// ---- DUTs/Sensirion/ST_SensirionFMStatus.TcDUT
TYPE ST_SensirionFMStatus :
STRUCT
	

	iFlowTicks	:	INT;
	uiSensorOutput	: UINT;
	iState	:	INT;
	rFlow	:	REAL; // units of uL/min
	xOoR	:	BOOL; // Out of range
	xFMMode :	BOOL; // calib mode 0 = prec, 1 = extended
	xFlowValid	:	BOOL; // driver completes successfully
	abReply	:	ARRAY[1..500] OF BYTE;
	bAdr	:	BYTE; //Device address
	bStatus	:	BYTE; //Sensor status
(* Bit 0: 0: Sensor idle
		1: Sensor Busy
Bit 1: 	0: Continuous Measurement disabled
		1: Continuous Measurement enabled
Bit 2: (for Firmware . 1.3)
		0: Auto detection Measurement disabled
		1: Auto detection Measurement enabled
Bit 3: (for Firmware . 1.3)
		0: No Auto Measurement since last read out Status
		1: Auto Measurement finished since last read out Status, is set back to 0 after read out *)

END_STRUCT
END_TYPE

// ---- DUTs/ST_M3GasManifold.TcDUT
TYPE ST_M3GasManifold :
STRUCT
	stManiVlv1	:	ST_ManifoldValve;
	stManiVlv2	:	ST_ManifoldValve;
	stManiVlv3	:	ST_ManifoldValve;
	stManiVlv4	:	ST_ManifoldValve;
	stManiVlv5	:	ST_ManifoldValve;
	stManiVlv6	:	ST_ManifoldValve;
	stManiVlv7	:	ST_ManifoldValve;
	stManiVlv8	:	ST_ManifoldValve;
	
	xOnline	:	BOOL; //WC inverse (true is good)
END_STRUCT
END_TYPE

// ---- DUTs/ST_Proportionair.TcDUT
TYPE ST_Proportionair :
STRUCT
	
(* Control *)
xEnable	:	BOOL;
iSetpoint	:	INT;
iSetpointRaw	:	INT;
iHiLimit	:	INT;
iLoLimit	:	INT;

(* Readback *)
xStable	:	BOOL;//TTL signal from the proportionair controller that the pressure is stable
iPressure	:	INT;
iPressureRaw : INT;


END_STRUCT
END_TYPE

// ---- DUTs/ST_Selector.TcDUT
TYPE ST_Selector :
STRUCT

	(* Meta info *)
	iId	: INT;	// Used to ID the selector attached to the system
	(* iId: Implemented to support switching selectors on the fly,
	the ID tells us which flow meter code to use, as the M2
	used several different flowmeters. *)

	(* Flowmeter *)
	(* Declare a structure for every possible FM *)
	stSelFMStatusBh	:	ST_BhFMStatus;
	stSelFMStatusSens	:	ST_SensirionFMStatus;
	stSelFMControlBh	:	ST_BhFMControl;
	stSelFMControlSens	:	ST_SensirionFMControl;
		
	
	//Common parameters
	iFlowMeterType	:	INT; //see below
	(*  1 = Sensirion
		2 = Bronkhorst
	*)
	
	xFMReset : BOOL; // Pulse only.
	rFlow : REAL; //uL/min
	xFMOoR	:	BOOL; // Out of range (too high)
	xFlowValid	:	BOOL; // driver completes successfully
	xFMModeReq	:	BOOL; //for sensirion calibration range (request)
	xFMModeRb	:	BOOL; //for sensirion calibration range (readback)
	(*
	field(ZRST, "OK")
	field(ONST, "OoR>")
	field(TWST, "<OoR")
	field(THST, "Flow Invalid")
	*)
	iFMState	:	INT;

	(* Selector controls *)
	xResLock	:	BOOL; // request to lock the valves
	xResUnlock	:	BOOL; // request to unlock the valves
	xResLocked	:	BOOL; // valve movement is locked
	xResSyncd	:	BOOL; // valves are on the same position
	iSyncReqPos	:	INT;
	iVici1ReqPos : INT;
	iVici2ReqPos : INT;
	stViciVlvCtrl	: ARRAY[1..2] OF	ST_ViciControl;
	
	
	(* Selector Readbacks *)
	iSyncResPos : INT;
	stViciVlvStatus	: ARRAY[1..2] OF	ST_ViciStatus;
	
	(* Shakers *)
	stShaker01	:	ST_Shaker;
	stShaker02	:	ST_Shaker;
	stShaker03	:	ST_Shaker;
	stShaker04	:	ST_Shaker;
	

END_STRUCT
END_TYPE

// ---- DUTs/ST_ShakerControls.TcDUT
TYPE ST_ShakerControls :
STRUCT
	
xShaker1On	:	BOOL;
xShaker2On	:	BOOL;
xShaker3On	:	BOOL;
xShaker4On	:	BOOL;
xShaker5On	:	BOOL;
xShaker6On	:	BOOL;
xShaker7On	:	BOOL;
xShaker8On	:	BOOL;

END_STRUCT
END_TYPE

// ---- DUTs/Vici/ST_ViciControl.TcDUT
TYPE ST_ViciControl :
STRUCT
	sViciReply			: STRING;
	iReqPos				: INT;
	xDirection			:BOOL;
	iAddress				:INT;
END_STRUCT
END_TYPE

// ---- GVLs/GVL.TcGVL
VAR_GLOBAL
 mb_Input_Coils   : ARRAY [0..255] OF BOOL;
 mb_Output_Coils : ARRAY [0..255] OF BOOL;
 mb_Input_Registers : ARRAY [0..255] OF WORD;
 mb_Output_Registers : ARRAY [0..255] OF WORD;
 
 mb_PLC_Memory	AT	%MW0	:	ARRAY[0..1000] OF WORD;
 
 	g_xFirstPass: BOOL := TRUE;
	g_xIOState	:	BOOL := FALSE;
	g_aEcatMaster1 AT %I* : AMSNETID;
	g_aEcatMaster2 AT %I* : AMSNETID;
	

 
END_VAR

// ---- GVLs/GVL_Autosave.TcGVL
VAR_GLOBAL PERSISTENT
	
	gp_stWaterRegDeadband	:	ST_RegDeadbandControls;
	gp_stSheathRegDeadband	:	ST_RegDeadbandControls;

	gp_stSelector	:	ST_Selector;
	gp_stSelector2	:	ST_Selector;
	
	gp_stRegProp1	:	ST_Proportionair;
	gp_stRegProp2	:	ST_Proportionair;
	gp_stRegProp3	:	ST_Proportionair;
	gp_stRegProp4	:	ST_Proportionair;

END_VAR

// ---- GVLs/GVL_ComBuffers.TcGVL
VAR_GLOBAL
	
	SerialRXBuffer_SelVici : ComBuffer;
	SerialTXBuffer_SelVici : ComBuffer;
	
	SerialRXBuffer_SelFlwMtr : ComBuffer;
	SerialTXBuffer_SelFlwMtr : ComBuffer;
	
	SerialRXBuffer_Sel2FlwMtr : ComBuffer;
	SerialTXBuffer_Sel2FlwMtr : ComBuffer;
	
	SerialRXBuffer_Sel2Vici : ComBuffer;
	SerialTXBuffer_Sel2Vici : ComBuffer;
	
	SerialRXBuffer_CoolerShakerTEC : ComBuffer;
	SerialTXBuffer_CoolerShakerTEC : ComBuffer;
	
END_VAR

// ---- GVLs/GVL_Devices.TcGVL
VAR_GLOBAL
	
	(* Selector*)
	stSelector	:	ST_Selector;
	stSelector2	:	ST_Selector;
	
	(* Cooler shaker *)
	stTECCtrl	: ARRAY[1..3] OF	ST_TECControl;
	stTECStatus	: ARRAY[1..3] OF	ST_TECStatus;
	
	stRegProp1	:	ST_Proportionair;
	stRegProp2	:	ST_Proportionair;
	stRegProp3	:	ST_Proportionair;
	stRegProp4	:	ST_Proportionair;
	
	(* Shakers *)
	stShaker01	:	ST_Shaker;
	stShaker02	:	ST_Shaker;
	stShaker03	:	ST_Shaker;
	stShaker04	:	ST_Shaker;
	
	(* Minitti Manifold *)
	stGasMani	:	ST_M3GasManifold;
	
	(* ALI *)
	stALI	:	ST_ALI;

END_VAR

// ---- GVLs/GVL_IO.TcGVL
VAR_GLOBAL
	
	iq_stM2SelectorA	:	ST_M2SelectorIO;
	iq_stM2SelectorB	:	ST_M2SelectorIO;

	iq_stM3SelectorA	:	ST_M3SelectorIO;
	iq_stM3SelectorB	:	ST_M3SelectorIO;
	
	iq_stPressCtrlA		:	ST_M3PressCtrlIO;
	iq_stPressCtrlB		:	ST_M3PressCtrlIO;

	i_iFscEB1Ch0AI	AT	%I*	:	INT;
	i_iFscEB1Ch1AI	AT	%I*	:	INT;
	i_iFscEB1Ch2AI	AT	%I*	:	INT;
	i_iFscEB1Ch3AI	AT	%I*	:	INT;
	
	iq_stM3GasManifold	:	ST_M3GasManifoldIO;

END_VAR

// ---- Version/Global_Version.TcGVL
// This function has been automatically generated from the project information.
VAR_GLOBAL CONSTANT
	{attribute 'const_non_replaced'}
	stLibVersion_SDS_M2 : ST_LibVersion := (iMajor := 2, iMinor := 6, iBuild := 0, iRevision := -1, sVersion := '2.6.0');
END_VAR

// ---- POUs/MAIN.TcPOU
PROGRAM MAIN
VAR
	
		fb_S_UPS	:	FB_S_UPS;
		
		fbEcatDiag1	:	FB_EcatDiag;
		fbEcatDiag2 :	FB_EcatDiag;
	
END_VAR



//fb_S_UPS.iPLCPort := AMSPORT_R0_PLC_RTS2;
fb_S_UPS(iPLCPort:=851);


p_modbusRx();

p_Autosave();

p_ESTOP();

fbEcatDiag1(i_AMSNetId:=g_aEcatMaster1, i_xFirstPass:=g_xFirstPass, q_xAllStatesGood=>g_xIOState);
fbEcatDiag2(i_AMSNetId:=g_aEcatMaster2, i_xFirstPass:=g_xFirstPass, q_xAllStatesGood=>g_xIOState);

p_SoftIO();

//p_SelectorDetector();

p_SampleSelector();
p_SampleSelector2();
p_Regulators();
p_Manifold();
p_ALI();
//p_VacGaugeSup();


//p_CoolerShaker();

p_ModbusTx();

p_StatusLights();

(* Following execution of all the programs, set the first pass false *)
g_xFirstPass := FALSE;

END_PROGRAM

// ---- POUs/p_ModbusRx.TcPOU
PROGRAM p_ModbusRx
VAR
END_VAR

(* Modbus Controls from EPICS *)

(* General System Controls *)
xEnableRemoteControl := mb_Output_Coils[0];
g_xEstop		:= mb_Output_Coils[1];

IF xEnableRemoteControl THEN
xN2Purge	:= mb_Output_Coils[9];

(* Selector Controls *)
stSelector.iVici1ReqPos := mb_Output_Registers[30];
stSelector.iVici2ReqPos := mb_Output_Registers[31];
stSelector.iSyncReqPos	:= mb_Output_Registers[32];

stSelector.xResLock := mb_Output_Coils[30];
stSelector.xFMReset := mb_Output_Coils[31];
stSelector.xFMModeReq 	:= mb_Output_Coils[32];
stSelector.xResUnlock := mb_Output_Coils[33];

stSelector.stShaker01.i_xEpics := mb_Output_Coils[10];
stSelector.stShaker02.i_xEpics := mb_Output_Coils[11];
stSelector.stShaker03.i_xEpics := mb_Output_Coils[12];
stSelector.stShaker04.i_xEpics := mb_Output_Coils[13];

(* Selector 2 Controls *)
stSelector2.iVici1ReqPos := mb_Output_Registers[40];
stSelector2.iVici2ReqPos := mb_Output_Registers[41];
stSelector2.iSyncReqPos	:= mb_Output_Registers[42];

stSelector2.xResLock := mb_Output_Coils[40];
stSelector2.xFMReset := mb_Output_Coils[41];
stSelector2.xFMModeReq 	:= mb_Output_Coils[42];
stSelector2.xResUnlock := mb_Output_Coils[43];

stSelector2.stShaker01.i_xEpics := mb_Output_Coils[44];
stSelector2.stShaker02.i_xEpics := mb_Output_Coils[45];
stSelector2.stShaker03.i_xEpics := mb_Output_Coils[46];
stSelector2.stShaker04.i_xEpics := mb_Output_Coils[47];

(* Proportionair controls *)
stRegProp1.xEnable:=mb_Output_Coils[50];  //Proportionair controls
stRegProp2.xEnable:=mb_Output_Coils[51];  //Proportionair controls

stRegProp3.xEnable:=mb_Output_Coils[52];  //Proportionair controls
stRegProp4.xEnable:=mb_Output_Coils[53];  //Proportionair controls

stRegProp1.iSetpoint:=mb_Output_Registers[50];  //Proportionair controls
stRegProp2.iSetpoint:=mb_Output_Registers[51];  //Proportionair controls
stRegProp1.iHiLimit:=mb_Output_Registers[52];  //Proportionair controls
stRegProp2.iHiLimit:=mb_Output_Registers[53];  //Proportionair controls

stRegProp3.iSetpoint:=mb_Output_Registers[54];  //Proportionair controls
stRegProp4.iSetpoint:=mb_Output_Registers[55];  //Proportionair controls
stRegProp3.iHiLimit:=mb_Output_Registers[56];  //Proportionair controls
stRegProp4.iHiLimit:=mb_Output_Registers[57];  //Proportionair controls

(* Digital output controls *)
stManiVlv1.xSW:=mb_Output_Coils[60];  //Minitti manifold valve controls
stManiVlv2.xSW:=mb_Output_Coils[61];  //Minitti manifold valve controls
stManiVlv3.xSW:=mb_Output_Coils[62];  //Minitti manifold valve controls
stManiVlv4.xSW:=mb_Output_Coils[63];  //Minitti manifold valve controls
stManiVlv5.xSW:=mb_Output_Coils[64];  //Minitti manifold valve controls
stManiVlv6.xSW:=mb_Output_Coils[65];  //Minitti manifold valve controls
stManiVlv7.xSW:=mb_Output_Coils[66];  //Minitti manifold valve controls
stManiVlv8.xSW:=mb_Output_Coils[67];  //Minitti manifold valve controls
//=========================================================
// ALI Controls
	stALI.axisX.xStart:=mb_Output_Coils[80];  //ALI_Manip
	stALI.axisX.xStop:=mb_Output_Coils[81];  //ALI_Manip
	stALI.axisY.xStart:=mb_Output_Coils[82];  //ALI_Manip
	stALI.axisY.xStop:=mb_Output_Coils[83];  //ALI_Manip
	stALI.axisZ.xStart:=mb_Output_Coils[84];  //ALI_Manip
	stALI.axisZ.xStop:=mb_Output_Coils[85];  //ALI_Manip
	
	stALI.stPropVlv.xEnable := mb_Output_Coils[86];
	
	stALI.axisX.xReset:=mb_Output_Coils[87];  //ALI_Manip
	stALI.axisY.xReset:=mb_Output_Coils[88];  //ALI_Manip
	stALI.axisZ.xReset:=mb_Output_Coils[89];  //ALI_Manip
	
	stALI.stPropVlv.i_iPercOpenSP := mb_Output_Registers[80]; //ALI Propvalve
	stALI.stPropVlv.ePVCtrlStateReq := mb_Output_Registers[81]; //ALI Propvalve
	MEMCPY(srcAddr:=ADR(mb_PLC_Memory[90]), destAddr:=ADR(stALI.axisX.rReqAbsPos), n:=SIZEOF(stALI.axisX.rReqAbsPos)); //ALI CTRL
	MEMCPY(srcAddr:=ADR(mb_PLC_Memory[92]), destAddr:=ADR(stALI.axisY.rReqAbsPos), n:=SIZEOF(stALI.axisY.rReqAbsPos)); //ALI CTRL
	MEMCPY(srcAddr:=ADR(mb_PLC_Memory[94]), destAddr:=ADR(stALI.axisZ.rReqAbsPos), n:=SIZEOF(stALI.axisZ.rReqAbsPos)); //ALI CTRL
	MEMCPY(srcAddr:=ADR(mb_PLC_Memory[96]), destAddr:=ADR(stALI.stPropVlv.i_rPressSP), n:=SIZEOF(stALI.stPropVlv.i_rPressSP)); //ALI CTRL

END_IF

END_PROGRAM

// ---- POUs/p_Autosave.TcPOU
PROGRAM p_Autosave
VAR
END_VAR

(* If first pass, copy all persistent variables (which should be intialized to old values) back into the operational variables *)
IF g_xFirstPass THEN
	
	stRegProp1 := gp_stRegProp1;
	stRegProp2 := gp_stRegProp2;
	stRegProp3 := gp_stRegProp3;
	stRegProp4 := gp_stRegProp4;
	
ELSE
	gp_stRegProp1 := stRegProp1;
	gp_stRegProp2 := stRegProp2;
	gp_stRegProp3 := stRegProp3;
	gp_stRegProp4 := stRegProp4;
	
END_IF

END_PROGRAM

// ---- POUs/p_ESTOP.TcPOU
PROGRAM p_ESTOP
VAR
	rtEstop : R_TRIG;
END_VAR

(* 
Estop checks for a rising edge on the estop global variable then triggeres the following actions
1. Set selector to position 12, the default resting place
2. Set the water regulator to 0
The sheath regulator is not set to zero at this point because we don't want to ice the jet.
*)

rtEstop(CLK:=g_xEstop);

(* Check for E-Stop *)
IF rtEstop.Q THEN
	stSelector.iVici1ReqPos := 12;
	stSelector.iVici2ReqPos := 12;
	stSelector.iSyncReqPos	:= 12;	
END_IF

END_PROGRAM

// ---- POUs/p_SoftIO.TcPOU
PROGRAM p_SoftIO
VAR
END_VAR

(* Shakers *)
stSelector.stShaker01.i_xSwitch := iq_stM2SelectorA.i_EP2338_Ch5;
stSelector.stShaker02.i_xSwitch := iq_stM2SelectorA.i_EP2338_Ch6;
stSelector.stShaker03.i_xSwitch := iq_stM2SelectorA.i_EP2338_Ch7;
stSelector.stShaker04.i_xSwitch := iq_stM2SelectorA.i_EP2338_Ch8;

iq_stM2SelectorA.q_EP2338_Ch1	:= stSelector.stShaker01.q_xPwrDO;
iq_stM2SelectorA.q_EP2338_Ch2	:= stSelector.stShaker02.q_xPwrDO;
iq_stM2SelectorA.q_EP2338_Ch3	:= stSelector.stShaker03.q_xPwrDO;
iq_stM2SelectorA.q_EP2338_Ch4	:= stSelector.stShaker04.q_xPwrDO;

stSelector2.stShaker01.i_xSwitch := iq_stM2SelectorB.i_EP2338_Ch5;
stSelector2.stShaker02.i_xSwitch := iq_stM2SelectorB.i_EP2338_Ch6;
stSelector2.stShaker03.i_xSwitch := iq_stM2SelectorB.i_EP2338_Ch7;
stSelector2.stShaker04.i_xSwitch := iq_stM2SelectorB.i_EP2338_Ch8;

iq_stM2SelectorB.q_EP2338_Ch1	:= stSelector2.stShaker01.q_xPwrDO;
iq_stM2SelectorB.q_EP2338_Ch2	:= stSelector2.stShaker02.q_xPwrDO;
iq_stM2SelectorB.q_EP2338_Ch3	:= stSelector2.stShaker03.q_xPwrDO;
iq_stM2SelectorB.q_EP2338_Ch4	:= stSelector2.stShaker04.q_xPwrDO;

stRegProp1.iPressureRaw := iq_stPressCtrlA.i_EP4374_Ch1;
stRegProp2.iPressureRaw := iq_stPressCtrlA.i_EP4374_Ch2;

iq_stPressCtrlA.q_EP4374_Ch3 := stRegProp1.iSetpointRaw;
iq_stPressCtrlA.q_EP4374_Ch4 := stRegProp2.iSetpointRaw;

stRegProp3.iPressureRaw := iq_stPressCtrlB.i_EP4374_Ch1;
stRegProp4.iPressureRaw := iq_stPressCtrlB.i_EP4374_Ch2;

iq_stPressCtrlB.q_EP4374_Ch3 := stRegProp3.iSetpointRaw;
iq_stPressCtrlB.q_EP4374_Ch4 := stRegProp4.iSetpointRaw;

END_PROGRAM

// ---- POUs/p_Regulators.TcPOU
PROGRAM p_Regulators
VAR

fbRegProp1	:	FB_ProportionairRegulator;
fbRegProp2	:	FB_ProportionairRegulator;
fbRegProp3	:	FB_ProportionairRegulator;
fbRegProp4	:	FB_ProportionairRegulator;

END_VAR

(* Proportionair regulators *)
fbRegProp1(iq_stRegProp:=stRegProp1);
fbRegProp2(iq_stRegProp:=stRegProp2);
fbRegProp3(iq_stRegProp:=stRegProp3);
fbRegProp4(iq_stRegProp:=stRegProp4);

END_PROGRAM

// ---- POUs/Regulators/FB_ProportionairRegulator.TcPOU
FUNCTION_BLOCK FB_ProportionairRegulator
VAR_INPUT
END_VAR
VAR_OUTPUT
END_VAR
VAR_IN_OUT
	iq_stRegProp	:	ST_Proportionair;
END_VAR
VAR
END_VAR

(* A. Wallace 2015-10-7
Proportionair regulator control *)

(* Pressure signal conversion, max pressure out 1000 (I think...) *)
iq_stRegProp.iPressure := REAL_TO_INT(1000 * (INT_TO_REAL(iq_stRegProp.iPressureRaw) / 32767));

iq_stRegProp.iSetpoint := LIMIT(iq_stRegProp.iLoLimit, iq_stRegProp.iSetpoint, iq_stRegProp.iHiLimit);

iq_stRegProp.iSetpointRaw := REAL_TO_INT( (INT_TO_REAL(iq_stRegProp.iSetpoint)/1000)*32767);

END_FUNCTION_BLOCK

// ---- POUs/p_Manifold.TcPOU
PROGRAM p_Manifold
VAR
	fbManiValve : FB_ManiValve;
END_VAR

(* Valve 1 *)
stManiVlv1.xILK := TRUE;
fbManiValve(iq_valve:=stManiVlv1);

(* Valve 2 *)
stManiVlv2.xILK := TRUE;
fbManiValve(iq_valve:=stManiVlv2);

(* Valve 3 *)
stManiVlv3.xILK := TRUE;
fbManiValve(iq_valve:=stManiVlv3);

(* Valve 4 *)
stManiVlv4.xILK := TRUE;
fbManiValve(iq_valve:=stManiVlv4);

(* Valve 5 *)
stManiVlv5.xILK := TRUE;
fbManiValve(iq_valve:=stManiVlv5);

(* Valve 6 *)
stManiVlv6.xILK := TRUE;
fbManiValve(iq_valve:=stManiVlv6);

(* Valve 7 *)
stManiVlv7.xILK := TRUE;
fbManiValve(iq_valve:=stManiVlv7);

(* Valve 8 *)
stManiVlv8.xILK := TRUE;
fbManiValve(iq_valve:=stManiVlv8);

END_PROGRAM

// ---- POUs/p_ALI.TcPOU
PROGRAM p_ALI
VAR
	fbALI_A	:	FB_ALI;
END_VAR

fbALI_A(iq_Injector:=stALI);

END_PROGRAM

// ---- POUs/ALI/FB_ALI.TcPOU
FUNCTION_BLOCK FB_ALI
VAR_IN_OUT
	iq_Injector	:	ST_ALI;
END_VAR
VAR_INPUT
END_VAR
VAR_OUTPUT
END_VAR
VAR
	fb925ALINB1 : FB_925;
	fb925ALINB2 : FB_925;
	fb722ALINB3 : FB_GCM;
	
	fbManipX	:	FB_ManipAxis;
	fbManipY	:	FB_ManipAxis;
	fbManipZ	:	FB_ManipAxis;
	

	
	fbPropValve		:	FB_PropValve;
	
	ftHotPlug	:	F_TRIG;
END_VAR

//When the system is plugged in, WC goes to zero, so reset motion control and other stuff
ftHotPlug(CLK:=iq_Injector.i_SyncUnitWC);

(* Soft IO *)
iq_Injector.stNozzleBoxVG.iPRESS_R :=iq_Injector.i_EP3174_Ch1;
iq_Injector.stSkimmerVG.iPRESS_R := iq_Injector.i_EP3174_Ch2;
iq_Injector.stRelaxVG.iPRESS_R := iq_Injector.i_EP3174_Ch3;

(* Vacuum Gauge Supervisor *)
fb925ALINB1(VG:=iq_Injector.stNozzleBoxVG);
fb925ALINB2(VG:=iq_Injector.stSkimmerVG);
fb722ALINB3(VG:=iq_Injector.stRelaxVG);

(* Butterfly valve *)
iq_Injector.stPropVlv.xInterlock := TRUE;
fbPropValve(stPropValve:=iq_Injector.stPropVlv, i_xExtIlk := TRUE);

(* Manipulator *)
fbManipX(iq_ManipAxis:=iq_Injector.axisX, i_xHotPlug:=ftHotPlug.Q);
fbManipY(iq_ManipAxis:=iq_Injector.axisY, i_xHotPlug:=ftHotPlug.Q);
fbManipZ(iq_ManipAxis:=iq_Injector.axisZ, i_xHotPlug:=ftHotPlug.Q);
F_AxisRef_To_MSTA(stManipAxis:=iq_Injector.axisX, MSTA=>iq_Injector.axisX.uiMsta);
F_AxisRef_To_MSTA(stManipAxis:=iq_Injector.axisY, MSTA=>iq_Injector.axisY.uiMsta);
F_AxisRef_To_MSTA(stManipAxis:=iq_Injector.axisZ, MSTA=>iq_Injector.axisZ.uiMsta);

END_FUNCTION_BLOCK

// ---- POUs/ALI/FB_ManipAxis.TcPOU
FUNCTION_BLOCK FB_ManipAxis
VAR_INPUT
	i_xHotPlug	:	BOOL;
END_VAR
VAR_OUTPUT
	q_asResult: ARRAY [1..20] OF STRING;
	q_xError	:	BOOL;
END_VAR
VAR_IN_OUT
	iq_ManipAxis	:	ST_ManipAxis;
END_VAR
VAR

	mcPower	:	MC_Power;
	mcReset	:	MC_Reset;
	mcMoveAbsolute : ARRAY[1..2] OF MC_MoveAbsolute;
	mcHalt	:	MC_Halt;
	mcSmoothMover	:	MC_SmoothMover;
	//Error Stuff
	indexResult: INT := 1;
	fbFormatString	:	FB_FormatString;
	
	xInitComplete	:	BOOL := FALSE;
	
	imcBlockIndex: INT;
	
	rtEnable : R_TRIG;
	ftEnable : F_TRIG;
	rtStop	:	R_TRIG;
	rtStart	:	R_TRIG;
	rReqAbsPosOld: REAL := 0;
	rReqAbsPosPrevious: REAL;
	iI: INT;
END_VAR

(* Manipulator Axis Function Block
Alex Wallace, 2016-8-8 

This block works by jumping between two absolute move blocks and buffering
the motion between them.
*)


rtEnable(CLK:=iq_ManipAxis.xEnable);
ftEnable(CLK:=iq_ManipAxis.xEnable);

//Update status
iq_ManipAxis.stAxis();

IF rtEnable.Q OR ftEnable.Q THEN
	xInitComplete := FALSE;
	iq_ManipAxis.eState := Init;
ELSIF xInitComplete THEN
	iq_ManipAxis.eState := MoveEnabled;
END_IF

//For EPICS, because the modbus map was made for 32 bit..
iq_ManipAxis.rActPos := LREAL_TO_REAL(iq_ManipAxis.stAxis.NcToPlc.ActPos);


CASE iq_ManipAxis.eState OF
	0: iq_ManipAxis.eState := Init;
	Init:
	(* Start by initializing the motor axis *)
	mcPower.Enable := iq_ManipAxis.xEnable;
	iq_ManipAxis.rReqAbsPos := iq_ManipAxis.rActPos; //do this when the PLC comes up so we don't just lose the position if we tweak
	IF mcPower.Status THEN //success
		xInitComplete := TRUE;
		q_asResult[indexResult] := 'Motor init success';
		indexResult := indexResult + 1;
		iq_ManipAxis.eState := MoveEnabled;
	ELSIF mcPower.Error THEN
		mcPower.Enable := FALSE;
		fbFormatString(sFormat:='Init mcPower Error: %s', arg1:=F_UDINT(mcPower.ErrorID));
		ActError();
	END_IF
		
	MoveEnabled:
		mcSmoothMover.Enable := iq_ManipAxis.xEnable;
		mcSmoothMover.ReqAbsPos := LIMIT(-100, REAL_TO_LREAL(iq_ManipAxis.rReqAbsPos), 100);
		mcSmoothMover.Execute := iq_ManipAxis.xStart;
		(*We've already captured the rising edge of start (if there was one, so 
		go ahead and reset it.*)
		iq_ManipAxis.xStart := FALSE;
		
		//Halt
		mcHalt.Execute S= iq_ManipAxis.xStop;
		mcHalt.Execute R= mcHalt.Busy;
		iq_ManipAxis.xStop R= mcHalt.Busy;
		IF mcPower.Error OR mcSmoothMover.Error THEN
			iq_ManipAxis.eState:=Error;
		END_IF
		
	Error:
		mcReset.Execute := rtEnable.Q OR i_xHotPlug OR iq_ManipAxis.xReset;
		IF mcReset.Done THEN
			q_xError := FALSE;
			mcReset.Execute := FALSE;
			iq_ManipAxis.xReset := FALSE;
			iq_ManipAxis.eState:=Init;
		END_IF
	
END_CASE


(* Run the mc blocks *)
ActPower();
mcReset(Axis:=iq_ManipAxis.stAxis);
mcSmoothMover(Axis:=iq_ManipAxis.stAxis,
	Velocity:=iq_ManipAxis.lrVelocity);
mcHalt(Axis:=iq_ManipAxis.stAxis);

iq_ManipAxis.xDmov := mcHalt.Done OR mcSmoothMover.Done;
iq_ManipAxis.xMovn := mcHalt.Busy OR mcSmoothMover.Busy;

//For display, this logic is not for safety
iq_ManipAxis.xHLS := NOT iq_ManipAxis.xHiLS;
iq_ManipAxis.xLLS := NOT iq_ManipAxis.xLoLS;

ACTION ActPower:
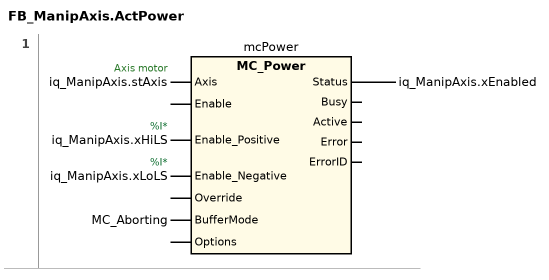
// NETWORK 1
//   iq_ManipAxis.stAxis: Axis motor
//   iq_ManipAxis.xHiLS: AT %I*
//   iq_ManipAxis.xLoLS: AT %I*
mcPower(
    Axis := iq_ManipAxis.stAxis,
    Enable_Positive := iq_ManipAxis.xHiLS,
    Enable_Negative := iq_ManipAxis.xLoLS,
    BufferMode := MC_Aborting); // MC_Power
iq_ManipAxis.xEnabled := mcPower.Status;
END_ACTION

ACTION ActError:
(* Error action
*)

//Reset the debugging index
IF indexResult > 20 THEN indexResult := 1; END_IF

iq_ManipAxis.eState := Error;
q_xError	:=	TRUE;
q_asResult[indexResult] := fbFormatString.sOut;
indexResult := indexResult +1;
END_ACTION

END_FUNCTION_BLOCK

// ---- POUs/ALI/MC_SmoothMover.TcPOU
FUNCTION_BLOCK MC_SmoothMover
VAR_IN_OUT
	Axis	:	AXIS_REF;
END_VAR
VAR_INPUT
	Velocity : LREAL;
	ReqAbsPos : LREAL; //A
	Enable	:	BOOL; //While true the block will accept new positions and attempt to move to them if they are different
	Execute	:	BOOL; //Will retry a move if the target position is the same
END_VAR
VAR_OUTPUT
	Done	:	BOOL;
	Busy	:	BOOL;
	Error	:	BOOL;
END_VAR
VAR
	mcMoveAbsolute : ARRAY[1..2] OF MC_MoveAbsolute;
	iI: INT;
	imcBlockIndex: INT;
	ReqAbsPosPrevious	: LREAL;
	rtExecute: R_TRIG;
END_VAR

(* Smooth Mover
2017-8-30
A. Wallace

Enable means the block will always aquire new positions as they are updated. Execute
can be used to retry a move.
*)


rtExecute(CLK:=Execute);

IF ( (ReqAbsPos <> ReqAbsPosPrevious AND Enable) OR rtExecute.Q) THEN
			mcMoveAbsolute[imcBlockIndex].Execute := FALSE;
			imcBlockIndex := imcBlockIndex + 1;
			IF imcBlockIndex >2 THEN imcBlockIndex := 1; END_IF
			mcMoveAbsolute[imcBlockIndex].Position := ReqAbsPos;
			mcMoveAbsolute[imcBlockIndex].Execute := TRUE;
			ReqAbsPosPrevious := ReqAbsPos;
		ELSIF mcMoveAbsolute[imcBlockIndex].Done OR 
				mcMoveAbsolute[imcBlockIndex].CommandAborted OR 
				mcMoveAbsolute[imcBlockIndex].Busy OR 
				mcMoveAbsolute[imcBlockIndex].Error THEN
			mcMoveAbsolute[imcBlockIndex].Execute := FALSE;
		END_IF
		
FOR iI := 1 TO 2 DO
	mcMoveAbsolute[iI](Axis := Axis, Velocity:=Velocity, BufferMode:=MC_Aborting);
END_FOR

Error := mcMoveAbsolute[1].Error OR mcMoveAbsolute[2].Error;
Done S= mcMoveAbsolute[1].Done OR mcMoveAbsolute[2].Done;
Busy := mcMoveAbsolute[1].Busy OR mcMoveAbsolute[2].Busy;
Done R= Busy OR Error;

END_FUNCTION_BLOCK

// ---- POUs/ALI/FB_PropValve.TcPOU
FUNCTION_BLOCK FB_PropValve
VAR_INPUT
	i_xExtIlk	:	BOOL;
END_VAR
VAR_OUTPUT
	q_xError	:	BOOL;
END_VAR
VAR_IN_OUT
	stPropValve	:	ST_PropValveMKS253;
END_VAR
VAR
	xInterlock	:	BOOL;
	
	eState : E_PropValveFBState := E_PropValveFBState.Init;
	stDiag	:	ST_fbDiagnostics;
	
	mcPower	:	MC_Power;
	mcJog	:	MC_Jog;
	mcReset	:	MC_Reset;
	mcSmoothMover	:	MC_SmoothMover;
	tofLLSFilter	:	TOF := (PT:=T#100MS);
	tofHLSFilter	:	TOF := (PT:=T#100MS);
	
	fbPID	:	FB_PID_EXT;
	
	AnyError: BOOL;
	xReady	:	BOOL;
	rtReset: R_TRIG;
	
	UpperLimit : LREAL := 2000;
END_VAR

(* Provide the motor enable and limit switch functions for the MKS 253 valve *)

xInterlock := stPropValve.xInterlock AND i_xExtIlk;
stPropValve.xEnable R= NOT xInterlock;


rtReset(CLK:=stPropValve.xEnable);

(* The low limit switch was flakey, I added the filters *)
tofLLSFilter(IN:=stPropValve.i_LLS);
tofHLSFilter(IN:=stPropValve.i_HLS);
mcPower.Enable_Positive := tofHLSFilter.Q;
mcPower.Enable_Negative := tofLLSFilter.Q;
mcPower.Enable := xInterlock AND stPropValve.xEnable;
stPropValve.xEnabled := mcPower.Enable;
(* Move the valve *)

IF AnyError THEN
	eState := E_PropValveFBState.Error;
	stPropValve.ePVCtrlStateReq := HMI_PropValveCtrlState.Hold;
ELSIF xReady THEN
	CASE stPropValve.ePVCtrlStateReq OF
		HMI_PropValveCtrlState.Hold:
			eState := E_PropValveFBState.Hold;
		HMI_PropValveCtrlState.Manual:
			eState := E_PropValveFBState.Manual;
		HMI_PropValveCtrlState.Pressure:
			eState := E_PropValveFBState.Pressure;
	END_CASE
ELSE
	eState := E_PropValveFBState.Init;
END_IF

CASE eState OF
	E_PropValveFBState.Init:
		//This state is reached at startup and after a reset
		//It seeks the closed limit switch and moves to hold
		stPropValve.ePVCtrlState := HMI_PropValveCtrlState.Hold;
		fbPID.i_Reset := TRUE;
		IF NOT tofLLSFilter.Q AND mcPower.Status THEN
			stPropValve.ePVCtrlStateReq := HMI_PropValveCtrlState.Hold;
			fbPID.i_Reset := TRUE;
			xReady := TRUE;
		END_IF
	E_PropValveFBState.Hold:
		stPropValve.ePVCtrlState := HMI_PropValveCtrlState.Hold;
		mcJog.JogForward := FALSE;
		mcJog.JogBackwards := FALSE;
		fbPID.i_Hold := TRUE;
		
	E_PropValveFBState.Pressure:
		stPropValve.ePVCtrlState := HMI_PropValveCtrlState.Pressure;
		
		fbPID.i_Hold := FALSE;
		fbPID.i_Reset := FALSE;
		
		//If the PID output is positive, jog forward, velocity scaled by the PID output
		//likewise for a negative PID output
		mcJog.JogForward := fbPID.q_lrCtrlOutput > 0;
		mcJog.JogBackwards := fbPID.q_lrCtrlOutput < 0;
		mcJog.Velocity := ABS(fbPID.q_lrCtrlOutput) * stPropValve.lrMaxSpeed;
		
	E_PropValveFBState.Manual:
		stPropValve.ePVCtrlState := HMI_PropValveCtrlState.Manual;
		fbPID.i_Hold := TRUE;
		mcSmoothMover.Enable := TRUE;
		mcSmoothMover.ReqAbsPos := LIMIT(0, INT_TO_LREAL(stPropValve.i_iPercOpenSP), 100)/100*UpperLimit;
		
	E_PropValveFBState.Error:
		//Purgatory
		mcJog.JogBackwards := FALSE;
		mcJog.JogForward  := FALSE;
		fbPID.i_Hold := TRUE;
		xReady	:= FALSE;
END_CASE


//Valve movement based on PID output
fbPID(i_lrSetpoint := REAL_TO_LREAL(stPropValve.i_rPressSP),
		i_lrActVal := REAL_TO_LREAL(stPropValve.i_rPressRB),
		i_stPIDParams := stPropValve.stPIDParams);
	
	
//MC blocks	
mcPower(Axis:=stPropValve.stAxis);	
mcReset(Axis:=stPropValve.stAxis);
mcJog(Axis:=stPropValve.stAxis, Mode:=E_JogMode.MC_JOGMODE_CONTINOUS);
mcSmoothMover(Axis:=stPropValve.stAxis, 
		Velocity:=stPropValve.lrMaxSpeed); 

AnyError := mcJog.Error OR mcPower.Error OR fbPID.q_Error OR mcSmoothMover.Error;

(* EPICS display of perc open *)
stPropValve.q_iPercOpen := LREAL_TO_INT(100*stPropValve.stAxis.NcToPlc.ActPos / UpperLimit);

(* EPICS display of limits *)
stPropValve.xHLS := NOT tofHLSFilter.Q;
stPropValve.xLLS := NOT tofLLSFilter.Q;

END_FUNCTION_BLOCK

// ---- POUs/ALI/FB_PID_EXT.TcPOU
FUNCTION_BLOCK FB_PID_EXT
VAR_INPUT
	i_lrSetpoint	:	LREAL;
	i_lrActVal	:	LREAL;
	i_stPIDParams	:	ST_PIDParams;
	//Hold the output and pause the block
	i_Hold	:	BOOL;
	i_Reset	:	BOOL;
END_VAR
VAR_OUTPUT
	q_lrCtrlOutput	:	LREAL;
	q_Error	:	BOOL;
	q_Limited	:	BOOL;
END_VAR
VAR
	fbPID	:	FB_BasicPID;
	eState	:	E_CTRL_MODE;
	xInitialized	:	BOOL := FALSE;
	lrSetpoint	:	LREAL;
	lrActVal	:	LREAL;
	bReset: BOOL;
	lrCtrlOutput: LREAL;
	xFirstPass: BOOL;
	stDiag	:	ST_fbDiagnostics;
END_VAR

(*

NOTE: If the PID block is having issues check the cycle time, it might be wrong.
*)
IF fbPID.nErrorStatus <> 0 THEN
	eState := E_CTRL_MODE.Error;
ELSIF fbPID.nErrorStatus = 0 AND xInitialized THEN
	q_Error := FALSE;
	IF i_Hold THEN 
		eState := E_CTRL_MODE.Hold;
	ELSE
		eState := E_CTRL_MODE.Run;
	END_IF
END_IF

CASE eState OF
	E_CTRL_MODE.Init:
		//Complete 1 pass through this FB to check PID block for errors
		IF xFirstPass THEN
			xInitialized := FALSE;//pass
		ELSE
			xInitialized := TRUE;
		END_IF
	E_CTRL_MODE.Run:
		lrSetpoint := i_lrSetpoint;
		lrCtrlOutput := fbPID.fCtrlOutput;
		bReset := FALSE;
	E_CTRL_MODE.Hold:
	(* While holding, the setpoint value is set to the actual
	value and the execution of the PID block is paused *)
		lrSetpoint := lrActVal;
		lrCtrlOutput := lrCtrlOutput;
		bReset := TRUE;
	E_CTRL_MODE.Error:
		q_Error := TRUE;
		lrSetpoint := 0;
		lrCtrlOutput := 0;
END_CASE

fbPID(fSetpointValue := lrSetpoint,
	fActualValue := lrActVal,
	bReset := bReset,
	fCtrlCycleTime :=i_stPIDParams.fCtrlCycleTime,
	fKp := i_stPIDParams.fKp,
	fTn := i_stPIDParams.fTn,
	fTv := i_stPIDParams.fTv,
	fTd := i_stPIDParams.fTd
	);

//Hold everything until fb is initialized
IF xInitialized AND NOT q_Error THEN
	//Indicate that the output is being limited
	q_Limited := lrCtrlOutput > i_stPIDParams.fUpperLim OR lrCtrlOutput < i_stPIDParams.fLowerLim;
	q_lrCtrlOutput := LIMIT(i_stPIDParams.fLowerLim, lrCtrlOutput, i_stPIDParams.fUpperLim);
ELSE
	q_lrCtrlOutput := 0;
	q_Limited := FALSE;
END_IF

xFirstPass := False;

END_FUNCTION_BLOCK

// ---- POUs/ALI/F_AxisRef_To_MSTA.TcPOU
FUNCTION F_AxisRef_To_MSTA	: UINT
VAR_INPUT
	stManipAxis	:	ST_ManipAxis;
END_VAR
VAR_OUTPUT
	MSTA	:	UINT;
END_VAR
VAR
END_VAR

(* This block translates the axis ref status to an EPICS psuedo MSTA value *)
(* A. Wallace, 17/8/17 *)

MSTA.1 := stManipAxis.stAxis.Status.Error;
MSTA.0 := stManipAxis.xEnabled;

END_FUNCTION

// ---- POUs/p_ModbusTx.TcPOU
PROGRAM p_ModbusTx
VAR
END_VAR

(* Modbus controls/ readbacks back to EPICS *)

(* Global system controls *)
mb_Input_Coils[0] := xEnableRemoteControl;
mb_Input_Coils[1] := xSystemPressurized;

mb_Input_Coils[10]:=iq_stPressCtrlA.i_SyncUnitWC;  //WC readbacks
mb_Input_Coils[11]:=iq_stPressCtrlB.i_SyncUnitWC;  //WC readbacks
mb_Input_Coils[12]:=iq_stM2SelectorA.i_SyncUnitWC;  //WC readbacks
mb_Input_Coils[13]:=iq_stM2SelectorB.i_SyncUnitWC;  //WC readbacks
mb_Input_Coils[14]:=iq_stM3SelectorA.i_SyncUnitWC;  //WC readbacks
mb_Input_Coils[15]:=iq_stM3SelectorB.i_SyncUnitWC;  //WC readbacks
mb_Input_Coils[16]:=stAli.i_SyncUnitWC;

(* Selector Controls *)
mb_Output_Registers[30] := stSelector.iVici1ReqPos;
mb_Output_Registers[31] := stSelector.iVici2ReqPos;
mb_Output_Registers[32] := stSelector.iSyncReqPos;
mb_Output_Coils[30] := 0;
mb_Output_Coils[31]:= stSelector.xFMReset;
mb_Output_Coils[33] := 0;

(* Selector 2 Controls *)
mb_Output_Registers[40] := stSelector2.iVici1ReqPos;
mb_Output_Registers[41] := stSelector2.iVici2ReqPos;
mb_Output_Registers[42] := stSelector2.iSyncReqPos;
mb_Output_Coils[40] := stSelector2.xResLock;
mb_Output_Coils[41]:= stSelector2.xFMReset;

(* Selector Readbacks *)
mb_Input_Registers[30] := stSelector.stViciVlvStatus[1].iCurrPos;
mb_Input_Registers[31] := stSelector.stViciVlvStatus[2].iCurrPos;
mb_Input_Registers[32] := stSelector.iSyncResPos;
mb_Input_Registers[33] := stSelector.iFMState;
mb_Input_Registers[34] := stSelector.iFlowMeterType;

mb_Input_Coils[30] := stSelector.xFMOoR;
mb_Input_Coils[31] := stSelector.xFlowValid;
mb_Input_Coils[32] := stSelector.xResSyncd;
mb_Input_Coils[33] := stSelector.xResLocked;
mb_Input_Coils[34] := stSelector.xFMModeRb;

(* Selector 2 Readbacks *)
mb_Input_Registers[40] := stSelector2.stViciVlvStatus[1].iCurrPos;
mb_Input_Registers[41] := stSelector2.stViciVlvStatus[2].iCurrPos;
mb_Input_Registers[42] := stSelector2.iSyncResPos;
mb_Input_Registers[43] := stSelector2.iFMState;
mb_Input_Registers[44] := stSelector2.iFlowMeterType;

mb_Input_Coils[40] := stSelector2.xFMOoR;
mb_Input_Coils[41] := stSelector2.xFlowValid;
mb_Input_Coils[42] := stSelector2.xResSyncd;
mb_Input_Coils[43] := stSelector2.xResLocked;
mb_Input_Coils[44] := stSelector2.xFMModeRb;


(* Flow meters *)
MEMCPY(destAddr:=ADR( mb_PLC_Memory[0]), srcAddr:=ADR(stSelector.rFlow), n:=4);
MEMCPY(destAddr:=ADR( mb_PLC_Memory[16]), srcAddr:=ADR(stSelector2.rFlow), n:=4);

(* Proportionair controls *)
mb_Output_Coils[50]:=stRegProp1.xEnable;  //Proportionair controls
mb_Output_Coils[51]:=stRegProp2.xEnable;  //Proportionair controls

mb_Output_Coils[52]:=stRegProp3.xEnable;  //Proportionair controls
mb_Output_Coils[53]:=stRegProp4.xEnable;  //Proportionair controls

mb_Output_Registers[50]:=stRegProp1.iSetpoint;  //Proportionair controls
mb_Output_Registers[51]:=stRegProp2.iSetpoint;  //Proportionair controls
mb_Output_Registers[52]:=stRegProp1.iHiLimit;  //Proportionair controls
mb_Output_Registers[53]:=stRegProp2.iHiLimit;  //Proportionair controls

mb_Output_Registers[54]:=stRegProp3.iSetpoint;  //Proportionair controls
mb_Output_Registers[55]:=stRegProp4.iSetpoint;  //Proportionair controls
mb_Output_Registers[56]:=stRegProp3.iHiLimit;  //Proportionair controls
mb_Output_Registers[57]:=stRegProp4.iHiLimit;  //Proportionair controls

mb_Input_Registers[50]:=stRegProp1.iPressure;  //Proportionair readbacks
mb_Input_Registers[51]:=stRegProp2.iPressure;  //Proportionair readbacks

mb_Input_Registers[52]:=stRegProp3.iPressure;  //Proportionair readbacks
mb_Input_Registers[53]:=stRegProp4.iPressure;  //Proportionair readbacks

mb_Input_Coils[50]:=stRegProp1.xStable;  //Proportionair readbacks
mb_Input_Coils[51]:=stRegProp2.xStable;  //Proportionair readbacks

mb_Input_Coils[52]:=stRegProp3.xStable;  //Proportionair readbacks
mb_Input_Coils[53]:=stRegProp4.xStable;  //Proportionair readbacks


(* Minitti Manifold Controls *)
mb_Input_Coils[60]:=stGasMani.stManiVlv1.xILK;  //Minitti manifold valve controls
mb_Input_Coils[61]:=stGasMani.stManiVlv2.xILK;  //Minitti manifold valve controls
mb_Input_Coils[62]:=stGasMani.stManiVlv3.xILK;  //Minitti manifold valve controls
mb_Input_Coils[63]:=stGasMani.stManiVlv4.xILK;  //Minitti manifold valve controls
mb_Input_Coils[64]:=stGasMani.stManiVlv5.xILK;  //Minitti manifold valve controls
mb_Input_Coils[65]:=stGasMani.stManiVlv6.xILK;  //Minitti manifold valve controls
mb_Input_Coils[66]:=stGasMani.stManiVlv7.xILK;  //Minitti manifold valve controls
mb_Input_Coils[67]:=stGasMani.stManiVlv8.xILK;  //Minitti manifold valve controls
mb_Input_Coils[68]:=stGasMani.stManiVlv1.ixOPN;  //Minitti manifold valve controls
mb_Input_Coils[69]:=stGasMani.stManiVlv2.ixOPN;  //Minitti manifold valve controls
mb_Input_Coils[70]:=stGasMani.stManiVlv3.ixOPN;  //Minitti manifold valve controls
mb_Input_Coils[71]:=stGasMani.stManiVlv4.ixOPN;  //Minitti manifold valve controls
mb_Input_Coils[72]:=stGasMani.stManiVlv5.ixOPN;  //Minitti manifold valve controls
mb_Input_Coils[73]:=stGasMani.stManiVlv6.ixOPN;  //Minitti manifold valve controls
mb_Input_Coils[74]:=stGasMani.stManiVlv7.ixOPN;  //Minitti manifold valve controls
mb_Input_Coils[75]:=stGasMani.stManiVlv8.ixOPN;  //Minitti manifold valve controls
//=========================================================
// ALI Controls
	mb_Input_Coils[80]:=stALI.axisX.xHLS;  //ALI_Manip
	mb_Input_Coils[81]:=stALI.axisX.xLLS;  //ALI_Manip
	mb_Input_Coils[82]:=stALI.axisY.xHLS;  //ALI_Manip
	mb_Input_Coils[83]:=stALI.axisY.xLLS;  //ALI_Manip
	mb_Input_Coils[84]:=stALI.axisZ.xHLS;  //ALI_Manip
	mb_Input_Coils[85]:=stALI.axisZ.xLLS;  //ALI_Manip
	mb_Input_Coils[86]:=stALI.stPropVlv.xHLS;  //ALI_Manip
	mb_Input_Coils[87]:=stALI.stPropVlv.xLLS;  //ALI_Manip
	mb_Input_Coils[88]:=stALI.stPropVlv.xEnabled;  //ALI_Manip
	mb_Input_Coils[89]:=stALI.stPropVlv.xInterlock;  //ALI_Manip
	
	mb_Input_Coils[90]:=stALI.axisX.xMovn;  //ALI_Manip
	mb_Input_Coils[91]:=stALI.axisX.xDmov;  //ALI_Manip
	mb_Input_Coils[92]:=stALI.axisY.xMovn;  //ALI_Manip
	mb_Input_Coils[93]:=stALI.axisY.xDmov;  //ALI_Manip
	mb_Input_Coils[94]:=stALI.axisZ.xMovn;  //ALI_Manip
	mb_Input_Coils[95]:=stALI.axisZ.xDmov;  //ALI_Manip
	
	mb_Input_Registers[80]:=stALI.stPropVlv.q_iPercOpen;  //ALI_Manip
	mb_Input_Registers[81]:=stALI.axisX.uiMsta;  //ALI_Manip
	mb_Input_Registers[82]:=stALI.axisY.uiMsta;  //ALI_Manip
	mb_Input_Registers[83]:=stALI.axisZ.uiMsta;  //ALI_Manip
	mb_Input_Registers[84]:=stALI.stPropVlv.ePVCtrlState;  //ALI_Manip
	mb_Input_Registers[85]:=0;  //ALI_Manip
	mb_Input_Registers[86]:=0;  //ALI_Manip
	mb_Input_Registers[87]:=0;  //ALI_Manip
	mb_Input_Registers[88]:=0;  //ALI_Manip
	mb_Input_Registers[89]:=0;  //ALI_Manip
	
	mb_Output_Coils[80]:=stALI.axisX.xStart;  //ALI_Manip
	mb_Output_Coils[81]:=stALI.axisX.xStop;  //ALI_Manip
	mb_Output_Coils[82]:=stALI.axisY.xStart;  //ALI_Manip
	mb_Output_Coils[83]:=stALI.axisY.xStop;  //ALI_Manip
	mb_Output_Coils[84]:=stALI.axisZ.xStart;  //ALI_Manip
	mb_Output_Coils[85]:=stALI.axisZ.xStop;  //ALI_Manip
	mb_Output_Coils[86]:=stALI.stPropVlv.xEnable;  //ALI_Manip
	mb_Output_Coils[87]:=stALI.axisX.xReset;  //ALI_Manip
	mb_Output_Coils[88]:=stALI.axisY.xReset;  //ALI_Manip
	mb_Output_Coils[89]:=stALI.axisZ.xReset;  //ALI_Manip
	
	mb_Output_Registers[80]:=stALI.stPropVlv.i_iPercOpenSP;  //ALI_Manip
	mb_Output_Registers[81]:=stALI.stPropVlv.ePVCtrlStateReq;  //ALI_Manip
	mb_Output_Registers[82]:=0;  //ALI_Manip
	mb_Output_Registers[83]:=0;  //ALI_Manip
	mb_Output_Registers[84]:=0;  //ALI_Manip
	mb_Output_Registers[85]:=0;  //ALI_Manip
	mb_Output_Registers[86]:=0;  //ALI_Manip
	mb_Output_Registers[87]:=0;  //ALI_Manip
	mb_Output_Registers[88]:=0;  //ALI_Manip
	mb_Output_Registers[89]:=0;  //ALI_Manip
	
	MEMCPY(destAddr:=ADR(mb_PLC_Memory[70]), srcAddr:=ADR(stALI.axisX.rActPos), n:=SIZEOF(stALI.axisX.rActPos));  //ALI RB
	MEMCPY(destAddr:=ADR(mb_PLC_Memory[72]), srcAddr:=ADR(stALI.axisY.rActPos), n:=SIZEOF(stALI.axisY.rActPos));  //ALI RB
	MEMCPY(destAddr:=ADR(mb_PLC_Memory[74]), srcAddr:=ADR(stALI.axisZ.rActPos), n:=SIZEOF(stALI.axisZ.rActPos));  //ALI RB
	MEMCPY(destAddr:=ADR(mb_PLC_Memory[76]), srcAddr:=ADR(stALI.stSkimmerVG.rPRESS), n:=SIZEOF(stALI.stSkimmerVG.rPRESS));  //ALI RB
	MEMCPY(destAddr:=ADR(mb_PLC_Memory[78]), srcAddr:=ADR(stALI.stNozzleBoxVG.rPRESS), n:=SIZEOF(stALI.stNozzleBoxVG.rPRESS));  //ALI RB
	MEMCPY(destAddr:=ADR(mb_PLC_Memory[80]), srcAddr:=ADR(stALI.stRelaxVG.rPRESS), n:=SIZEOF(stALI.stRelaxVG.rPRESS));  //ALI RB
	MEMCPY(destAddr:=ADR(mb_PLC_Memory[90]), srcAddr:=ADR(stALI.axisX.rReqAbsPos), n:=SIZEOF(stALI.axisX.rReqAbsPos));  //ALI CTRL
	MEMCPY(destAddr:=ADR(mb_PLC_Memory[92]), srcAddr:=ADR(stALI.axisY.rReqAbsPos), n:=SIZEOF(stALI.axisY.rReqAbsPos));  //ALI CTRL
	MEMCPY(destAddr:=ADR(mb_PLC_Memory[94]), srcAddr:=ADR(stALI.axisZ.rReqAbsPos), n:=SIZEOF(stALI.axisZ.rReqAbsPos));  //ALI CTRL

END_PROGRAM

// ---- POUs/p_StatusLights.TcPOU
PROGRAM p_StatusLights
VAR
END_VAR

gxRedLight := xEnableRemoteControl;//Remote control in use
gxYellowLight := stRegSheath.wInPress > 100 OR stRegWater.wInPress > 100;
gxGreenLight := NOT (gxRedLight or gxYellowLight); (* attach system error or something here someday *)

END_PROGRAM

// ---- POUs/Bronkhorst/FB_L01Driver.TcPOU
FUNCTION_BLOCK FB_L01Driver

VAR_INPUT
	i_xExecute				: BOOL;					(* rising edge execute *)
	i_tTimeOut				: TIME := t#10s;  		(* Maximum wait time for reply *)
	i_stControl				: ST_BhFMControl;
END_VAR
VAR_OUTPUT
	q_xDone					: BOOL;
	q_xError				: BOOL;
	q_xWarning				: BOOL;					(* set in the event of an unexpected reply *)
	q_xTimeout				: BOOL;
	q_sResult				: STRING(255);
	q_sLastSentString		: ARRAY[1..40] OF STRING;				(* Last String Sent to Serial Device - for debugging *)
	q_sLastReceivedString	: ARRAY[1..40] OF STRING;				(* Last String Received from Serial Device - for debugging *)
	q_stStatus				: ST_BhFMStatus;
END_VAR
VAR_IN_OUT
	iq_stSerialRXBuffer 	: ComBuffer;
	iq_stSerialTXBuffer 	: ComBuffer;
END_VAR
VAR
	rtExecute				: R_TRIG;
	iStep					: INT;
	sSendData				: STRING;
	fbFlowBusTransaction		: FB_FlowBusTransaction;
	(*fbFormatString			: FB_FormatString;*)
	(*fbSplit					: FB_Split255;*)
	asReplyFields			: ARRAY[1..20] OF T_MaxString;
	wChecksum: WORD;

	sWorking: STRING;
	strResponseExpected: STRING;
END_VAR

(* This function block performs serial communication with a Bronkhorst L01 u-Flow meter *)

(* rising edge trigger *)
rtExecute(CLK:= i_xExecute);
IF rtExecute.Q  THEN
	q_xDone	:= FALSE;
	q_xError := FALSE;
	q_xWarning := FALSE;
	q_xTimeout := FALSE;
	q_sResult:= '';
	fbFlowBusTransaction( i_xExecute:= FALSE, iq_stSerialRXBuffer:= iq_stSerialRXBuffer, iq_stSerialTXBuffer:= iq_stSerialTXBuffer );  (* reset *)
	iStep := 10;
END_IF

CASE iStep OF
	0: (* idle *)
		;

	10: (* Get Flow *)
		fbFlowBusTransaction(
			i_xExecute:= TRUE,
			i_sNode:='80',
			i_sCmd:= '01',
			i_sProcess := '01',
			i_sParameter := '20',
			i_tTimeOut:= i_tTimeOut,
			iq_stSerialRXBuffer:= iq_stSerialRXBuffer,
			iq_stSerialTXBuffer:= iq_stSerialTXBuffer,
			i_CmdFlag :=FALSE);
			
		IF fbFlowBusTransaction.q_xError THEN
			q_sResult := CONCAT('in Step 10 serial transaction failed with message: ', fbFlowBusTransaction.q_sResult);
			q_stStatus.xFlowValid := FALSE; (* used to signal an invalid readback or control exchange *)
			iStep := 9000;
		ELSIF fbFlowBusTransaction.q_xDone THEN
			q_stStatus.sReply := fbFlowBusTransaction.q_sResponseData;
			
			(* Parsing the response *)
			sWorking := MID(q_stStatus.sReply, 8, 11);
			sWorking := CONCAT('16#', sWorking);
			q_stStatus.uiFlowPercentageRaw := STRING_TO_UINT(sWorking);
			q_stStatus.rFlowPercentage := UINT_TO_REAL(q_stStatus.uiFlowPercentageRaw) /32000;
			//Real flow
			q_stStatus.rFlow := (q_stStatus.rFlowPercentage * (2-0)(*g/h*) + 0(*g/h*)) * (1000(*uL*)/60(*min*));
			
			IF (q_stStatus.rFlow > 33(* uL/min *) ) THEN
				q_stStatus.iState := 1;
			ELSIF (q_stStatus.rFlow < 16 (* uL/min *) ) THEN
				q_stStatus.iState := 2;
			ELSE
				q_stStatus.iState := 0; //flow OK
			END_IF
			
			
			
			fbFlowBusTransaction( i_xExecute:= FALSE, iq_stSerialRXBuffer:= iq_stSerialRXBuffer, iq_stSerialTXBuffer:= iq_stSerialTXBuffer, i_CmdFlag :=FALSE);  (* reset *)
			iStep := 8000;
			
		END_IF


	8000: (* done *)
		q_xDone := TRUE;
		IF q_sResult = '' THEN
			q_sResult := 'Success';
		END_IF
		IF  i_xExecute = FALSE THEN
			q_xDone:= FALSE;
			iStep := 0;
		END_IF
		

	9000:
		_A_ClearStatus();
		q_xTimeout := fbFlowBusTransaction.q_xTimeout;
		q_xError := TRUE;
		q_stStatus.xFlowValid := FALSE;
		q_stStatus.iState := 3; //flow invalid

END_CASE

q_sLastSentString := fbFlowBusTransaction.q_sLastSentString;
q_sLastReceivedString := fbFlowBusTransaction.q_sLastReceivedString;

ACTION _A_ClearStatus:
q_stStatus.sReply := '';
END_ACTION

END_FUNCTION_BLOCK

// ---- POUs/FB_SelectorM3.TcPOU
FUNCTION_BLOCK FB_SelectorM3
VAR_INPUT
END_VAR
VAR_OUTPUT
END_VAR
VAR_IN_OUT
	iq_stSelector	:	ST_SelectorM3;
END_VAR
VAR
	fbSelectorSync	:	FB_SelectorSync;
	
	afbViciDriver : ARRAY [1..4] OF FB_ViciDriver;
	
	fbSensirionDriver	:	ARRAY [1..2] OF	FB_SensirionDriver;
	

	stStatus: STRING;
	udCount: UDINT;

	tofReset: TOF;

	iIdOld	:	INT;
	
	viciIndex: INT := 1;
	fmIndex: INT;
END_VAR

//Flowmeters
//////////////////////////////////////
Sensirion();

//Valve control
///////////////////////////////////
	fbSelectorSync(iq_stSelector:=iq_stSelector);
	iq_stSelector.stViciVlvCtrl[1].iReqPos := LIMIT(1, iq_stSelector.iVici1ReqPos, 12);
	iq_stSelector.stViciVlvCtrl[2].iReqPos := LIMIT(1, iq_stSelector.iVici2ReqPos, 12);
	ViciDrivers();

	//for epics readback to be consistent
	IF iq_stSelector.xResSyncd THEN iq_stSelector.iSyncResPos := iq_stSelector.stViciVlvStatus[1].iCurrPos; END_IF

(* Shakers *)
iq_stSelector.stShaker01.q_xPwrDO := iq_stSelector.stShaker01.i_xEpics;
iq_stSelector.stShaker02.q_xPwrDO := iq_stSelector.stShaker02.i_xEpics;
iq_stSelector.stShaker03.q_xPwrDO := iq_stSelector.stShaker03.i_xEpics;
iq_stSelector.stShaker04.q_xPwrDO := iq_stSelector.stShaker04.i_xEpics;

ACTION ViciDrivers:
afbViciDriver[viciIndex](
	i_xExecute:= TRUE,
	i_tTimeOut:= t#10s,
	i_stControl:= stSelector.stViciVlvCtrl[viciIndex],
	iq_stSerialRXBuffer:= SerialRXBuffer_SelVici,
	iq_stSerialTXBuffer:= SerialTXBuffer_SelVici,
	q_stStatus=>stSelector.stViciVlvStatus[viciIndex]);

IF 	afbViciDriver[viciIndex].q_xDone OR
	afbViciDriver[viciIndex].q_xError OR
	afbViciDriver[viciIndex].q_xTimeout THEN
	(* reset function for next time *)
	afbViciDriver[viciIndex](i_xExecute:=FALSE, iq_stSerialRXBuffer:= SerialRXBuffer_SelVici, iq_stSerialTXBuffer:=  SerialTXBuffer_SelVici);
	
	viciIndex := viciIndex + 1;
	IF viciIndex > 2 THEN viciIndex := 1; END_IF
	
END_IF
END_ACTION

ACTION Sensirion:
(* Sensirion Flowmeter driver encapsulation*)	

(* Reinitialize flowmeter *)
iq_stSelector[1].stSelFMControlSens.xReset := stSelector.xFMReset;
iq_stSelector[1].stSelFMControlSens.xCalMode := stSelector.xFMModeReq;

	
iq_stSelector.fbSensirionDriver[fmIndex](
	i_xExecute:= TRUE,
	i_tTimeOut:= t#10s,
	iq_stSerialRXBuffer:= SerialRXBuffer_SelFlwMtr,
	iq_stSerialTXBuffer:= SerialTXBuffer_SelFlwMtr,
	q_stStatus=>iq_stSelector.astSelFM[fmIndex].stat,
	i_stControl:=iq_stSelector.astSelFM[fmIndex].ctrl);

IF iq_stSelector.fbSensirionDriver[fmIndex].q_xDone OR
	iq_stSelector.fbSensirionDriver[fmIndex].q_xError OR
	iq_stSelector.fbSensirionDriver[fmIndex].q_xTimeout THEN

	//Legacy flow
	iq_stSelector.rFlow := iq_stSelector[fmIndex].stSelFMStatusSens.rFlow;
	iq_stSelector.xFMOoR := iq_stSelector[fmIndex].stSelFMStatusSens.xOoR;
	iq_stSelector.xFlowValid := iq_stSelector[fmIndex].stSelFMStatusSens.xFlowValid;
	iq_stSelector.iFMState := iq_stSelector[fmIndex].stSelFMStatusSens.iState;
	iq_stSelector.xFMModeRb := iq_stSelector[fmIndex].stSelFMStatusSens.xFMMode;
	
	//M3 flows
	iq_stSelector.rLowFlow := iq_stSelector[fmIndex].stSelFMStatusSens.rFlow;
	iq_stSelector.rHighFlow := iq_stSelector[fmIndex].stSelFMStatusSens.rFlow;
	
	(* reset function for next time *)
	iq_stSelector.fbSensirionDriver[fmIndex](i_xExecute:=FALSE, iq_stSerialRXBuffer:= SerialRXBuffer_SelFlwMtr, iq_stSerialTXBuffer:=  SerialTXBuffer_SelFlwMtr);

	fmIndex := fmIndex + 1;
	IF fmIndex > 2 THEN fmIndex := 1;	END_IF
END_IF
END_ACTION

END_FUNCTION_BLOCK

// ---- POUs/Helpers/FB_SelectorSync.TcPOU
FUNCTION_BLOCK FB_SelectorSync
VAR_INPUT
END_VAR
VAR_OUTPUT
END_VAR
VAR_IN_OUT
	iq_stSelector	:	ST_SELECTOR;
END_VAR
VAR
	tofResSyncd : TOF;
	rtResLocked	:	R_TRIG;
	rsResLocked	:	RS;
	
	rtResLock : R_TRIG;
	rtResUnlock : R_TRIG;
END_VAR

(* Selector valve sync FB for vici valves *)



(* Check if both valves are in the same position *)
(* Should probably add something to the driver to check if we are in motion*)
tofResSyncd.IN := (iq_stSelector.stViciVlvStatus[1].iCurrPos = iq_stSelector.stViciVlvStatus[2].iCurrPos ) AND 
			(iq_stSelector.stViciVlvStatus[1].xPosValid  ) AND (iq_stSelector.stViciVlvStatus[1].xPosValid); (* Check for valid position rb *)

(* Delay the loss of ResSyncd so the valves can both be queried before overriding *)
(* Using a tof, but you can also check that both valves have been queried *)
tofResSyncd(PT:=T#10S);
iq_stSelector.xResSyncd := tofResSyncd.Q;

//Set, reset of valve lock
rtResLock(CLK:=iq_stSelector.xResLock);
rtResUnlock(CLK:=iq_stSelector.xResUnlock);
rsResLocked(set:=rtResLock.Q OR g_xFirstPass, reset1:=rtResUnlock.Q OR NOT iq_stSelector.xResSyncd);
iq_stSelector.xResLocked := rsResLocked.Q1;


(* If valve lock just became active, set the SyncReqPos to current locked position *)
rtResLocked(CLK:=iq_stSelector.xResLocked);
(*
IF rtResLocked.Q THEN 
	iq_stSelector.iSyncReqPos := iq_stSelector.iVici1ReqPos;
END_IF
*)
(* If valve lock active, match valve positions from the valve req that changes req number *)
IF iq_stSelector.xResLocked AND iq_stSelector.xResSyncd THEN
	IF iq_stSelector.iVici1ReqPos <> iq_stSelector.iSyncReqPos THEN
		iq_stSelector.iSyncReqPos := iq_stSelector.iVici1ReqPos;
		iq_stSelector.iVici2ReqPos := iq_stSelector.iVici1ReqPos;
	ELSIF iq_stSelector.iVici2ReqPos <> iq_stselector.iSyncReqPos THEN
		iq_stSelector.iSyncReqPos := iq_stSelector.iVici2ReqPos;
		iq_stSelector.iVici1ReqPos := iq_stSelector.iVici2ReqPos;
	END_IF
END_IF

iq_stSelector.xResLock := FALSE;
iq_stSelector.xResUnlock := False;

END_FUNCTION_BLOCK

// ---- POUs/VICI/FB_ViciDriver.TcPOU
FUNCTION_BLOCK FB_ViciDriver
FUNCTION_BLOCK FB_ViciDriver
VAR_INPUT
	i_xExecute				: BOOL;					(* rising edge execute *)
	i_tTimeOut				: TIME := t#10s;  		(* Maximum wait time for reply *)
	i_stControl				: ST_ViciControl;
END_VAR
VAR_OUTPUT
	q_xDone					: BOOL;
	q_xError				: BOOL;
	q_xWarning				: BOOL;					(* set in the event of an unexpected reply *)
	q_xTimeout				: BOOL;
	q_sResult				: STRING(255);
	q_sLastSentString		: ARRAY[1..40] OF STRING;				(* Last String Sent to Serial Device - for debugging *)
	q_sLastReceivedString	: ARRAY[1..40] OF STRING;				(* Last String Received from Serial Device - for debugging *)
	q_stStatus				: ST_ViciStatus;
END_VAR
VAR_IN_OUT
	iq_stSerialRXBuffer 	: ComBuffer;
	iq_stSerialTXBuffer 	: ComBuffer;
END_VAR
VAR
	rtExecute				: R_TRIG;
	iStep					: INT;
	sSendData				: STRING;
	fbViciTransaction		: FB_ViciTransaction;
	(*fbFormatString			: FB_FormatString;*)
	(*fbSplit					: FB_Split255;*)
	asReplyFields			: ARRAY[1..20] OF T_MaxString;
	wChecksum: WORD;
	rtStartIntegration: R_TRIG;
	rtEndReset: R_TRIG;

	sWorking: STRING;
	strResponseExpected: STRING;
END_VAR

(* This function block performs serial transactions with a Vici *)

(* rising edge trigger *)
rtExecute(CLK:= i_xExecute);
IF rtExecute.Q  THEN
	q_xDone	:= FALSE;
	q_xError := FALSE;
	q_xWarning := FALSE;
	q_xTimeout := FALSE;
	q_sResult:= '';
	FBViciTransaction( i_xExecute:= FALSE, iq_stSerialRXBuffer:= iq_stSerialRXBuffer, iq_stSerialTXBuffer:= iq_stSerialTXBuffer );  (* reset *)
	iStep := 10;
END_IF

CASE iStep OF
	0: (* idle *)
		;

	10: (* Get Position *)
		FBViciTransaction(
			i_xExecute:= TRUE,
			i_iAddress:=i_stControl.iAddress,
			i_sSendData:= 'CP', (*declared postion readback Vici command*)
			i_tTimeOut:= i_tTimeOut,
			iq_stSerialRXBuffer:= iq_stSerialRXBuffer,
			iq_stSerialTXBuffer:= iq_stSerialTXBuffer,
			i_CmdFlag :=FALSE);
		IF FBViciTransaction.q_xError THEN
			q_sResult := CONCAT('in Step 10 serial transaction failed with message: ', FBViciTransaction.q_sResult);
			q_stStatus.xPosValid := FALSE; (* used to signal an invalid readback or control exchange *)
			iStep := 9000;
		ELSIF FBViciTransaction.q_xDone THEN
			q_stStatus.sViciReply := FBViciTransaction.q_sResponseData;
			(* grab the left two characters, they should equal CP *)
			strResponseExpected := CONCAT(INT_TO_STRING( i_stControl.iAddress), 'CP');
			IF LEFT(q_stStatus.sViciReply, 3) <> strResponseExpected (*'1CP'*) THEN
				(*use q-s Result to specify error type*)
				q_sResult := CONCAT(CONCAT('in step 10 unexpected response recieved: ', LEFT(q_stStatus.sViciReply, 3)),CONCAT(' instead of: ', CONCAT(INT_TO_STRING( i_stControl.iAddress), 'CP')));
					q_xWarning := TRUE;
				(* If they don't equal CP, then error *)
				q_stStatus.xPosValid := FALSE; (* used to signal an invalid readback or control exchange *)
				iStep := 9000;
			(* else then grab the right two characters and convert to INT *)
			ELSE
			sWorking := RIGHT(q_stStatus.sViciReply, 2);
			q_stStatus.iCurrPos (* pass that INT to the q_stStatus.iCurrPos *) := STRING_TO_INT(sWorking);
			q_stStatus.xPosValid := TRUE;
			FBViciTransaction( i_xExecute:= FALSE, iq_stSerialRXBuffer:= iq_stSerialRXBuffer, iq_stSerialTXBuffer:= iq_stSerialTXBuffer, i_CmdFlag :=FALSE);  (* reset *)
			iStep := 5000;
			END_IF
		END_IF


	5000: (* Set position*)
		IF q_stStatus.iReqPos <> i_stControl.iReqPos THEN
			(*noah's code *)
			IF i_stControl.iReqPos > 12 OR i_stControl.iReqPos < 1 THEN
				q_sResult := CONCAT('in step 5000 port range exceeded: ',FBViciTransaction.q_sResponseData);
				i_stControl.iReqPos := LIMIT(1, i_stControl.iReqPos,12);
			ELSIF q_stStatus.iCurrPos > i_stControl.iReqPos THEN
				sSendData := CONCAT('CC', INT_TO_STRING(i_stControl.iReqPos));
			ELSE
				sSendData := CONCAT('CW', INT_TO_STRING(i_stControl.iReqPos));
			END_IF
			FBViciTransaction(
				i_xExecute:= TRUE,
				i_sSendData:= sSendData,
				i_tTimeOut:= i_tTimeOut,
				i_iAddress:=i_stControl.iAddress,
				iq_stSerialRXBuffer:= iq_stSerialRXBuffer,
				iq_stSerialTXBuffer:= iq_stSerialTXBuffer,
				i_CmdFlag:=TRUE);
			IF FBViciTransaction.q_xError THEN
				q_sResult := CONCAT('in Step 5000 serial transaction failed with message: ', FBViciTransaction.q_sResult);
				iStep := 9000;
			ELSIF FBViciTransaction.q_xDone THEN
				FBViciTransaction(
					 i_xExecute:= FALSE,
					iq_stSerialRXBuffer:= iq_stSerialRXBuffer,
					iq_stSerialTXBuffer:= iq_stSerialTXBuffer,
					i_CmdFlag:=FALSE );  (* reset *)
				q_stStatus.iReqPos := i_stControl.iReqPos;
				iStep := 8000;
			END_IF
		ELSE
			iStep := 8000;
		END_IF


	8000: (* done *)
		q_xDone := TRUE;
		IF q_sResult = '' THEN
			q_sResult := 'Success';
		END_IF
		IF  i_xExecute = FALSE THEN
			q_xDone:= FALSE;
			iStep := 0;
		END_IF

	9000:
		_A_ClearStatus();
		q_xTimeout := FBViciTransaction.q_xTimeout;
		q_xError := TRUE;
		

END_CASE

q_sLastSentString := FBViciTransaction.q_sLastSentString;
q_sLastReceivedString := FBViciTransaction.q_sLastReceivedString;

ACTION _A_ClearStatus:
q_stStatus.sViciReply := '';
END_ACTION

END_FUNCTION_BLOCK

// ---- POUs/VICI/FB_ViciTransaction.TcPOU
FUNCTION_BLOCK FB_ViciTransaction
VAR_INPUT
	i_xExecute				: BOOL;				(* Rising edge execute *)
	i_sSendData				: STRING; 			(* Send Data *)
	i_iAddress				:INT;
	i_tTimeOut				: TIME := t#10s;  	(* Maximum wait time for reply *)
	i_CmdFlag: BOOL := FALSE;
END_VAR
VAR_OUTPUT
	q_xDone					: BOOL;
	q_sResponseData			: STRING;
	q_xError				: BOOL;
	q_xTimeout				: BOOL;
	q_sResult				: STRING;
	q_sLastSentString		: ARRAY[1..40] OF STRING;			(* Last String Sent to Serial Device - for debugging *)
	q_sLastReceivedString	: ARRAY[1..40] OF STRING;			(* Last String Received from Serial Device - for debugging *)
END_VAR
VAR_IN_OUT
	iq_stSerialRXBuffer 	: ComBuffer;
	iq_stSerialTXBuffer 	: ComBuffer;
END_VAR
VAR
	rtExecute				: R_TRIG;
	iStep					: INT;
	fbClearComBuffer		: ClearComBuffer;
	fbSendString			: SendString;
	fbReceiveString			: ReceiveString;
	sReceivedString			: STRING;
	tonTimeout				: TON;
	sSendString: STRING;
	iStringTx: INT := 1;
	iStringRx: INT := 1;
	
	iStringTxRx: INT := 1;
	sTxRxString: ARRAY[1..40] OF STRING;
END_VAR

(* This function block performs serial transactions with a VICI *)

(* rising edge trigger *)
rtExecute(CLK:= i_xExecute);
IF rtExecute.Q THEN
	q_xDone	:= FALSE;
	q_sResponseData := '';
	q_xError := FALSE;
	q_xTimeout := FALSE;
	q_sResult:= '';
	q_sLastSentString[iStringTx] := '';
	q_sLastReceivedString[iStringRx]:= '';
	iStep := 10;
END_IF

CASE iStep OF
	0:
		; (* idle *)

	10: (* clear com buffers *)
		fbClearComBuffer(Buffer:= iq_stSerialRXBuffer);
		fbClearComBuffer(Buffer:= iq_stSerialTXBuffer);
		(* Reset receive *)
		fbReceiveString(
			Reset:= TRUE,
			ReceivedString:= sReceivedString,
			RXbuffer:= iq_stSerialRXBuffer );
		(* send the string *)
		sSendString := INT_TO_STRING(i_iAddress); (*building address header *)
		sSendString := CONCAT(sSendString, i_sSendData); (* adding the header *)
		sSendString := CONCAT(sSendString,'$R$L'); (* add <cr><lf> *) (*adding tail *)
		fbSendString( SendString:= sSendString, TXbuffer:= iq_stSerialTXBuffer );
		q_sLastSentString[iStringTx] := sSendString;
IF iStringTx = 40 THEN iStringTx := 1; ELSE iStringTx := iStringTx +1; END_IF
		iStep := iStep + 10;

	20: (* Finish sending the String *)
		IF fbSendString.Busy THEN
			fbSendString( SendString:= sSendString, TXbuffer:= iq_stSerialTXBuffer );
		ELSIF fbSendString.Error <> 0 THEN
			q_sResult := CONCAT('In step 20 fbSendString resulted in error: ', INT_TO_STRING(fbSendString.Error));
			iStep := 9000;
		ELSIF NOT fbSendString.Busy THEN
			(* if we are sending a position change request then we expect no reply *)
			IF i_CmdFlag THEN
				q_sResult := 'String sent....';
				q_xDone:= TRUE;
				iStep := 100;
			ELSE
				iStep:=iStep + 10;
			END_IF
		END_IF
		tonTimeout(IN:= FALSE);

	30: (* Get reply *)
		fbReceiveString(
			Prefix:= ,
			Suffix:= '$R',
			Timeout:= i_tTimeOut,
			Reset:= FALSE,
			ReceivedString:= sReceivedString,
			RXbuffer:= iq_stSerialRXBuffer );
		tonTimeout(IN:= TRUE, PT:= i_tTimeOut);
		IF fbReceiveString.Error <> 0 THEN
			q_sResult := CONCAT('In step 30 fbReceiveString resulted in error: ', INT_TO_STRING(fbReceiveString.Error));
			iStep := 9000;
		ELSIF fbReceiveString.RxTimeout OR tonTimeout.Q THEN
			q_sResult := 'Serial device failed to reply within timeout period';
			q_xTimeout := TRUE;
			iStep := 9000;
		ELSIF fbReceiveString.StringReceived THEN
			q_sLastReceivedString[iStringRx] := sReceivedString;
			IF iStringRx = 40 THEN iStringRx := 1; ELSE iStringRx := iStringRx +1; END_IF
			IF LEN(sReceivedString) < 2 THEN
				q_sResult := 'Reply too short.';
				iStep := 9000;
			ELSE
				q_sResponseData := LEFT(sReceivedString,LEN(sReceivedString)-1);
				q_sResult := 'Success.';
				q_xDone:= TRUE;
				iStep := 100;
				
			END_IF
		END_IF
		
		
		

	100: (* done *)
		IF  i_xExecute = FALSE THEN
			q_xDone:= FALSE;
			iStep := 0;
		END_IF
		IF NOT i_CmdFlag THEN
			sTxRxString[iStringTxRx]:=CONCAT(CONCAT(q_sLastSentString[iStringTx], ' received '), q_sLastReceivedString[iStringRx]);
		END_IF
		IF iStringTxRx = 40 THEN iStringTxRx := 1; ELSE iStringTxRx := iStringTxRx +1; END_IF

	9000:
		q_xError := TRUE;;




END_CASE

END_FUNCTION_BLOCK

// ---- POUs/Sensirion/FB_SensirionDriver.TcPOU
FUNCTION_BLOCK FB_SensirionDriver

VAR_INPUT
	i_xExecute				: BOOL;					(* rising edge execute *)
	i_tTimeOut				: TIME := T#10S;  		(* Maximum wait time for reply *)
	i_stControl				: ST_SensirionFMControl;
END_VAR
VAR_OUTPUT
	q_xDone					: BOOL;
	q_xError				: BOOL;
	q_xWarning				: BOOL;					(* set in the event of an unexpected reply *)
	q_xTimeout				: BOOL;
	q_asResult				: ARRAY[1..60] OF STRING(255);
	q_stStatus				: ST_SensirionFMStatus;
	q_xInitComplete			:	BOOL;
END_VAR
VAR_IN_OUT
	iq_stSerialRXBuffer 	: ComBuffer;
	iq_stSerialTXBuffer 	: ComBuffer;
END_VAR
VAR
	//Usual stuff
	rtExecute				: R_TRIG;
	rtReInit				:	R_TRIG;
	iStep					: INT;
	iResultIndex			:	INT := 1;
	aiSteps	:	ARRAY[1..256] OF INT;
	iStepIndex	:	INT;
	fbSensirionTransaction		: FB_SensirionTransaction;
	
	//Device Specific Working Variables
	tonDelay : TON;
	bLen	:	BYTE;
	abTxData	:	ARRAY[1..256] OF BYTE;
	xInitComplete	:	BOOL;
	abRxData	:	ARRAY[1..256] OF BYTE;
	
	iScale	:	INT;
	iUnit	:	INT;
	xType	:	BOOL;
	xMode	:	BYTE;
	xLinear	:	BOOL;
	uiOffset	:	UINT;
	iIdleAttempt : INT;
	
	//Command delays
	tonCommandDelay : TON;
xcatch : BOOL;
END_VAR

(* This function block performs serial communication with a Sensirion meter *)


(* 2015-4-8
The sensirion flow meter is direction agnostic. To make it work more like the Bronkhorst and other flowmeters
I limited the readback to the appropriate ranges. Negative flow is discarded.
*)

(* rising edge trigger *)
rtExecute(CLK:= i_xExecute);
rtReInit(CLK:= i_stControl.xReset);
IF rtReInit.Q THEN xInitComplete := FALSE; END_IF
IF rtExecute.Q  THEN
	q_xDone	:= FALSE;
	q_xError := FALSE;
	q_xWarning := FALSE;
	q_xTimeout := FALSE;
	q_asResult[iResultIndex]:= '';
	fbSensirionTransaction( i_xExecute:= FALSE, iq_stSerialRXBuffer:= iq_stSerialRXBuffer, iq_stSerialTXBuffer:= iq_stSerialTXBuffer );  (* reset *)
	IF xInitComplete THEN
		iStep := 30;
		(* Branch to reset device if reset bit is set here *)
		IF rtReInit.Q  OR (i_stControl.xCalMode <> q_stStatus.xFMMode) THEN
			iStep := 400;
			xInitComplete := FALSE;
			q_stStatus.xFlowValid := FALSE;
			q_asResult[iResultIndex] := 'Reinitializing';
			iResultIndex := iResultIndex +1;
		END_IF
	ELSIF i_stControl.xReset THEN
		iStep := 400;
		q_stStatus.xFlowValid := FALSE;
		q_asResult[iResultIndex] := 'Reinitializing';
		iResultIndex := iResultIndex +1;
	ELSE
		iStep := 9;
	END_IF
END_IF

CASE iStep OF
	0: (* idle *)
		;

	9: //Get cal mode
	fbSensirionTransaction(
		i_xExecute:= TRUE,
		i_bAdr:= q_stStatus.bAdr,
		i_bLen:= 0,
		i_bCmd:= 16#43,
		i_abTxData := abTxData,
		i_tTimeOut:= i_tTimeOut,
		iq_stSerialRXBuffer:= iq_stSerialRXBuffer,
		iq_stSerialTXBuffer:= iq_stSerialTXBuffer
		);
	IF fbSensirionTransaction.q_xError THEN
		q_asResult[iResultIndex] := CONCAT('in Step 9 serial transaction failed with message: ', fbSensirionTransaction.q_sResult);
		iResultIndex := iResultIndex +1;
		iStep := 9000;
	ELSIF fbSensirionTransaction.q_xDone THEN	
		//abRxdata := fbSensirionTransaction.q_baRxData;
		IF UDINT_TO_BOOL(MEMCPY(destAddr:=ADR(xMode), srcAddr:=ADR(fbSensirionTransaction.q_baRxData), n:=1)) THEN
			q_stStatus.xFMMode := BYTE_TO_BOOL(xMode);
			fbSensirionTransaction( i_xExecute:= FALSE, iq_stSerialRXBuffer:= iq_stSerialRXBuffer, iq_stSerialTXBuffer:= iq_stSerialTXBuffer );  (* reset *)
			q_asResult[iResultIndex] := CONCAT('Step 9 complete. Cal mode is set to: ', BYTE_TO_STRING(xMode));
			iResultIndex := iResultIndex +1;
		ELSE
			iStep := 9000;
			q_asResult[iResultIndex] := 'Memcpy in step 9 failed';
			iResultIndex := iResultIndex +1;
		END_IF
		iStep := 10;
	END_IF		
		
	10: // Set calibration
	//calibration of 0 for precision mode, 250 nL/min - 5000 nL/min
	// calibration of 1 for extended mode, 2000 nL/min - 20000 nL/min
	IF q_stStatus.xFMMode <> i_stControl.xCalMode THEN
		IF i_stControl.xCalMode THEN abTxData[1]:=1; ELSE abTxData[1]:=0; END_IF
		fbSensirionTransaction(
			i_xExecute:= TRUE,
			i_bAdr:= q_stStatus.bAdr,
			i_bLen:= 1,
			i_bCmd:= 16#43,
			i_abTxData := abTxData,
			i_tTimeOut:= i_tTimeOut,
			iq_stSerialRXBuffer:= iq_stSerialRXBuffer,
			iq_stSerialTXBuffer:= iq_stSerialTXBuffer
			);
		IF fbSensirionTransaction.q_xError THEN
			q_asResult[iResultIndex] := CONCAT('in Step 10 serial transaction failed with message: ', fbSensirionTransaction.q_sResult);
			iResultIndex := iResultIndex +1;
			iStep := 9000;
		ELSIF fbSensirionTransaction.q_xDone THEN
			tonCommandDelay(IN:=fbSensirionTransaction.q_xDone, PT:=T#1S);
			IF tonCommandDelay.Q THEN
				(* No response, completed transaction confirmed by a response*)
				q_asResult[iResultIndex] := 'Step 10 complete';
				iResultIndex := iResultIndex +1;
				iStep := 11;
				fbSensirionTransaction( i_xExecute:= FALSE, iq_stSerialRXBuffer:= iq_stSerialRXBuffer, iq_stSerialTXBuffer:= iq_stSerialTXBuffer );  (* reset *)
			END_IF
		END_IF
	ELSE
		q_asResult[iResultIndex] := 'Calmode already set';
		iResultIndex := iResultIndex +1;	
		iStep := 11;
	END_IF

	11: //Get cal mode
	fbSensirionTransaction(
		i_xExecute:= TRUE,
		i_bAdr:= q_stStatus.bAdr,
		i_bLen:= 0,
		i_bCmd:= 16#43,
		i_abTxData := abTxData,
		i_tTimeOut:= i_tTimeOut,
		iq_stSerialRXBuffer:= iq_stSerialRXBuffer,
		iq_stSerialTXBuffer:= iq_stSerialTXBuffer
		);
	IF fbSensirionTransaction.q_xError THEN
		q_asResult[iResultIndex] := CONCAT('in Step 11 serial transaction failed with message: ', fbSensirionTransaction.q_sResult);
		iResultIndex := iResultIndex +1;
		iStep := 9000;
	ELSIF fbSensirionTransaction.q_bState <> 0 THEN
		q_asResult[iResultIndex] := CONCAT('in Step 11 serial transaction failed with error state: ', BYTE_TO_STRING(fbSensirionTransaction.q_bState));
		iResultIndex := iResultIndex +1;
		fbSensirionTransaction( i_xExecute:= FALSE, iq_stSerialRXBuffer:= iq_stSerialRXBuffer, iq_stSerialTXBuffer:= iq_stSerialTXBuffer );  (* reset *)
		iStep := 9000;
	ELSIF fbSensirionTransaction.q_xDone THEN	
		tonCommandDelay(IN:=fbSensirionTransaction.q_xDone, PT:=T#100MS);
		IF tonCommandDelay.Q THEN
			IF UDINT_TO_BOOL(MEMCPY(destAddr:=ADR(xMode), srcAddr:=ADR(fbSensirionTransaction.q_baRxData), n:=1)) THEN
				q_stStatus.xFMMode := BYTE_TO_BOOL(xMode);
				fbSensirionTransaction( i_xExecute:= FALSE, iq_stSerialRXBuffer:= iq_stSerialRXBuffer, iq_stSerialTXBuffer:= iq_stSerialTXBuffer );  (* reset *)
				q_asResult[iResultIndex] := 'Step 11 complete';
				iResultIndex := iResultIndex +1;
				iStep := 12;
			ELSE
				iStep := 9000;
				q_asResult[iResultIndex] := 'Memcpy in step 9 failed';
				iResultIndex := iResultIndex +1;
			END_IF
		END_IF
	END_IF		
	
	12: //Get scale factor
	fbSensirionTransaction(
		i_xExecute:= TRUE,
		i_bAdr:= q_stStatus.bAdr,
		i_bLen:= 0,
		i_bCmd:= 16#53,
		i_abTxData := abTxData,
		i_tTimeOut:= i_tTimeOut,
		iq_stSerialRXBuffer:= iq_stSerialRXBuffer,
		iq_stSerialTXBuffer:= iq_stSerialTXBuffer
		);
	IF fbSensirionTransaction.q_xError THEN
		q_asResult[iResultIndex] := CONCAT('in Step 12 serial transaction failed with message: ', fbSensirionTransaction.q_sResult);
		iResultIndex := iResultIndex +1;
		iStep := 9000;
	ELSIF fbSensirionTransaction.q_bState <> 0 THEN
		q_asResult[iResultIndex] := CONCAT('in Step 12 serial transaction failed with error state: ', BYTE_TO_STRING(fbSensirionTransaction.q_bState));
		iResultIndex := iResultIndex +1;
		fbSensirionTransaction( i_xExecute:= FALSE, iq_stSerialRXBuffer:= iq_stSerialRXBuffer, iq_stSerialTXBuffer:= iq_stSerialTXBuffer );  (* reset *)
		iStep := 9000;
	ELSIF fbSensirionTransaction.q_xDone THEN	
		tonCommandDelay(IN:=fbSensirionTransaction.q_xDone, PT:=T#100MS);
		IF tonCommandDelay.Q THEN
			IF UDINT_TO_BOOL(MEMCPY(destAddr:=ADR(iScale), srcAddr:=ADR(fbSensirionTransaction.q_baRxData), n:=2)) THEN //always 2 for the 16 bit wide integer
				iScale := WORD_TO_INT(HOST_TO_BE16(INT_TO_WORD(iScale)));
				fbSensirionTransaction( i_xExecute:= FALSE, iq_stSerialRXBuffer:= iq_stSerialRXBuffer, iq_stSerialTXBuffer:= iq_stSerialTXBuffer );  (* reset *)
				q_asResult[iResultIndex] := 'Step 12 complete';
				iResultIndex := iResultIndex +1;
				iStep := 13;		
			ELSE
				iStep := 9000;
				q_asResult[iResultIndex] := 'Memcpy in step 12 failed';
				iResultIndex := iResultIndex +1;
			END_IF
		END_IF	
	END_IF
		
	13: //Get flow unit
	fbSensirionTransaction(
		i_xExecute:= TRUE,
		i_bAdr:= q_stStatus.bAdr,
		i_bLen:= 0,
		i_bCmd:= 16#52,
		i_abTxData := abTxData,
		i_tTimeOut:= i_tTimeOut,
		iq_stSerialRXBuffer:= iq_stSerialRXBuffer,
		iq_stSerialTXBuffer:= iq_stSerialTXBuffer
		);
	IF fbSensirionTransaction.q_xError THEN
		q_asResult[iResultIndex] := CONCAT('in Step 13 serial transaction failed with message: ', fbSensirionTransaction.q_sResult);
		iResultIndex := iResultIndex +1;
		iStep := 9000;
	ELSIF fbSensirionTransaction.q_bState <> 0 THEN
		q_asResult[iResultIndex] := CONCAT('in Step 13 serial transaction failed with error state: ', BYTE_TO_STRING(fbSensirionTransaction.q_bState));
		iResultIndex := iResultIndex +1;
		fbSensirionTransaction( i_xExecute:= FALSE, iq_stSerialRXBuffer:= iq_stSerialRXBuffer, iq_stSerialTXBuffer:= iq_stSerialTXBuffer );  (* reset *)
		iStep := 9000;
	ELSIF fbSensirionTransaction.q_xDone THEN	
		tonCommandDelay(IN:=fbSensirionTransaction.q_xDone, PT:=T#100MS);
		IF tonCommandDelay.Q THEN
			IF UDINT_TO_BOOL(MEMCPY(destAddr:=ADR(iUnit), srcAddr:=ADR(fbSensirionTransaction.q_baRxData), n:=2)) THEN //always 2 for the 16 bit wide integer
				iUnit := WORD_TO_INT(HOST_TO_BE16(INT_TO_WORD(iUnit)));
				fbSensirionTransaction( i_xExecute:= FALSE, iq_stSerialRXBuffer:= iq_stSerialRXBuffer, iq_stSerialTXBuffer:= iq_stSerialTXBuffer );  (* reset *)
				q_asResult[iResultIndex] := 'Step 13 complete';
				iResultIndex := iResultIndex +1;
				iStep := 14;
			ELSE
				iStep := 9000;
				q_asResult[iResultIndex] := 'Memcpy in step 13 failed';
				iResultIndex := iResultIndex +1;
			END_IF
		END_IF
	END_IF

	14: //Get measurement type
	fbSensirionTransaction(
		i_xExecute:= TRUE,
		i_bAdr:= q_stStatus.bAdr,
		i_bLen:= 0,
		i_bCmd:= 16#55,
		i_abTxData := abTxData,
		i_tTimeOut:= i_tTimeOut,
		iq_stSerialRXBuffer:= iq_stSerialRXBuffer,
		iq_stSerialTXBuffer:= iq_stSerialTXBuffer
		);
	IF fbSensirionTransaction.q_xError THEN
		q_asResult[iResultIndex] := CONCAT('in Step 14 serial transaction failed with message: ', fbSensirionTransaction.q_sResult);
		iResultIndex := iResultIndex +1;
		iStep := 9000;
	ELSIF fbSensirionTransaction.q_bState <> 0 THEN
		q_asResult[iResultIndex] := CONCAT('in Step 14 serial transaction failed with error state: ', BYTE_TO_STRING(fbSensirionTransaction.q_bState));
		iResultIndex := iResultIndex +1;
		fbSensirionTransaction( i_xExecute:= FALSE, iq_stSerialRXBuffer:= iq_stSerialRXBuffer, iq_stSerialTXBuffer:= iq_stSerialTXBuffer );  (* reset *)
		iStep := 9000;
	ELSIF fbSensirionTransaction.q_xDone THEN	
		tonCommandDelay(IN:=fbSensirionTransaction.q_xDone, PT:=T#100MS);
		IF tonCommandDelay.Q THEN
			xType := BYTE_TO_BOOL(fbSensirionTransaction.q_baRxData[1]);
			q_asResult[iResultIndex] := 'Step 14 complete';
			iResultIndex := iResultIndex +1;
			iStep := 16;
			fbSensirionTransaction( i_xExecute:= FALSE, iq_stSerialRXBuffer:= iq_stSerialRXBuffer, iq_stSerialTXBuffer:= iq_stSerialTXBuffer );  (* reset *)
		END_IF
	END_IF
	
	15: //Get offset
	fbSensirionTransaction(
		i_xExecute:= TRUE,
		i_bAdr:= q_stStatus.bAdr,
		i_bLen:= 0,
		i_bCmd:= 16#56,
		i_abTxData := abTxData,
		i_tTimeOut:= i_tTimeOut,
		iq_stSerialRXBuffer:= iq_stSerialRXBuffer,
		iq_stSerialTXBuffer:= iq_stSerialTXBuffer
		);
	IF fbSensirionTransaction.q_xError THEN
		q_asResult[iResultIndex] := CONCAT('in Step 15 serial transaction failed with message: ', fbSensirionTransaction.q_sResult);
		iResultIndex := iResultIndex +1;
		iStep := 9000;
	ELSIF fbSensirionTransaction.q_bState <> 0 THEN
		q_asResult[iResultIndex] := CONCAT('in Step 15 serial transaction failed with error state: ', BYTE_TO_STRING(fbSensirionTransaction.q_bState));
		iResultIndex := iResultIndex +1;
		fbSensirionTransaction( i_xExecute:= FALSE, iq_stSerialRXBuffer:= iq_stSerialRXBuffer, iq_stSerialTXBuffer:= iq_stSerialTXBuffer );  (* reset *)
		iStep := 9000;
	ELSIF fbSensirionTransaction.q_xDone THEN	
		tonCommandDelay(IN:=fbSensirionTransaction.q_xDone, PT:=T#100MS);
		IF tonCommandDelay.Q THEN
			IF UDINT_TO_BOOL(MEMCPY(destAddr:=ADR(uiOffset), srcAddr:=ADR(fbSensirionTransaction.q_baRxData), n:=2)) THEN //always 2 for the 16 bit wide integer
				uiOffset := WORD_TO_UINT(HOST_TO_BE16(UINT_TO_WORD(uiOffset)));
				A_ClearTransaction();  (* reset *)
				q_asResult[iResultIndex] := CONCAT('Step 15 complete, offset is: ', UINT_TO_STRING(uiOffset));
				iResultIndex := iResultIndex +1;
				iStep := 16;		
			ELSE
				iStep := 9000;
				q_asResult[iResultIndex] := 'Memcpy in step 15 failed';
				iResultIndex := iResultIndex +1;
			END_IF
			A_ClearTransaction();  (* reset *)
		END_IF
	END_IF
	
	16: //Get linear mode
	fbSensirionTransaction(
		i_xExecute:= TRUE,
		i_bAdr:= q_stStatus.bAdr,
		i_bLen:= 0,
		i_bCmd:= 16#45,
		i_abTxData := abTxData,
		i_tTimeOut:= i_tTimeOut,
		iq_stSerialRXBuffer:= iq_stSerialRXBuffer,
		iq_stSerialTXBuffer:= iq_stSerialTXBuffer
		);
	IF fbSensirionTransaction.q_xError THEN
		q_asResult[iResultIndex] := CONCAT('in Step 16 serial transaction failed with message: ', fbSensirionTransaction.q_sResult);
		iResultIndex := iResultIndex +1;
		iStep := 9000;
	ELSIF fbSensirionTransaction.q_bState <> 0 THEN
		q_asResult[iResultIndex] := CONCAT('in Step 16 serial transaction failed with error state: ', BYTE_TO_STRING(fbSensirionTransaction.q_bState));
		iResultIndex := iResultIndex +1;
		fbSensirionTransaction( i_xExecute:= FALSE, iq_stSerialRXBuffer:= iq_stSerialRXBuffer, iq_stSerialTXBuffer:= iq_stSerialTXBuffer );  (* reset *)
		iStep := 9000;
	ELSIF fbSensirionTransaction.q_xDone THEN	
		tonCommandDelay(IN:=fbSensirionTransaction.q_xDone, PT:=T#100MS);
		IF tonCommandDelay.Q THEN
			xLinear := BYTE_TO_BOOL(fbSensirionTransaction.q_baRxData[1]); 
			A_ClearTransaction();  (* reset *)
			q_asResult[iResultIndex] := CONCAT('Step 16 complete, linear is: ', BOOL_TO_STRING(xLinear));
			iResultIndex := iResultIndex +1;
			iStep := 20;		
		END_IF
	END_IF
	
//////////////////////////////////////////////////////////////////
// Reset sequence
//////////////////////////////////////////////////////////////////
(*
1. Issue a stop command to halt continuous measurement
2. Reset command
3. Reset initcomplete bit, and xReset
4. Move to done state
*)

	400: //Stop measurement
	fbSensirionTransaction(
		i_xExecute:= TRUE,
		i_bAdr:= q_stStatus.bAdr,
		i_bLen:= 0,
		i_bCmd:= 16#34,
		i_abTxData := abTxData,
		i_tTimeOut:= i_tTimeOut,
		iq_stSerialRXBuffer:= iq_stSerialRXBuffer,
		iq_stSerialTXBuffer:= iq_stSerialTXBuffer
		);
	IF fbSensirionTransaction.q_xError THEN
		q_asResult[iResultIndex] := CONCAT('in Step 400 serial transaction failed with message: ', fbSensirionTransaction.q_sResult);
		iResultIndex := iResultIndex +1;
		iStep := 9000;
	ELSIF fbSensirionTransaction.q_xDone THEN
		tonCommandDelay(IN:=fbSensirionTransaction.q_xDone, PT:=T#250MS);
		IF tonCommandDelay.Q THEN
			q_asResult[iResultIndex] := 'Measurement stop command sent';
			iResultIndex := iResultIndex +1;
			iStep:=405;
			fbSensirionTransaction( i_xExecute:= FALSE, iq_stSerialRXBuffer:= iq_stSerialRXBuffer, iq_stSerialTXBuffer:= iq_stSerialTXBuffer );  (* reset *)
		END_IF
	END_IF
	
	405: //Check sensor status
	fbSensirionTransaction(
		i_xExecute:= TRUE,
		i_bAdr:= q_stStatus.bAdr,
		i_bLen:= 0,
		i_bCmd:= 16#30,
		i_abTxData := abTxData,
		i_tTimeOut:= i_tTimeOut,
		iq_stSerialRXBuffer:= iq_stSerialRXBuffer,
		iq_stSerialTXBuffer:= iq_stSerialTXBuffer
		);
	IF fbSensirionTransaction.q_xError THEN
		q_asResult[iResultIndex] := CONCAT('in Step 405 serial transaction failed with message: ', fbSensirionTransaction.q_sResult);
		iResultIndex := iResultIndex +1;
		iStep := 9000;
	ELSIF fbSensirionTransaction.q_xDone THEN
		(* The status measurement is available at the rx data here *)
		IF fbSensirionTransaction.q_iRxLen > 0 THEN
			IF UDINT_TO_BOOL(MEMCPY(destAddr:=ADR(q_stStatus.bStatus), srcAddr:=ADR(fbSensirionTransaction.q_baRxData), n:=1)) THEN
				IF q_stStatus.bStatus.0 = 0 THEN //lsb of bStatus is idle
					iStep :=410;
					q_asResult[iResultIndex] := 'Sensor is idle.';
					iResultIndex := iResultIndex +1;
					fbSensirionTransaction( i_xExecute:= FALSE, iq_stSerialRXBuffer:= iq_stSerialRXBuffer, iq_stSerialTXBuffer:= iq_stSerialTXBuffer );  (* reset *)
				ELSE
					iStep := 400;
					iIdleAttempt := iIdleAttempt + 1;
					q_asResult[iResultIndex +1] := CONCAT('Failed to move to idle state in step 405, attempt ' , CONCAT(INT_TO_STRING(iIdleAttempt) , ' of 3'));
					IF iIdleAttempt = 3 THEN iStep := 9000; iIdleAttempt := 0; END_IF
					fbSensirionTransaction( i_xExecute:= FALSE, iq_stSerialRXBuffer:= iq_stSerialRXBuffer, iq_stSerialTXBuffer:= iq_stSerialTXBuffer );  (* reset *)
				END_IF
			ELSE
				iStep := 9000;
				q_asResult[iResultIndex] := 'Memcpy in step 405 failed';
				iResultIndex := iResultIndex +1;
			END_IF
		ELSE
			q_asResult[iResultIndex] := 'No status data returned';
			iResultIndex := iResultIndex +1;
			iStep := 9000;
		END_IF 		
	END_IF

	410: //Reset device
	fbSensirionTransaction(
		i_xExecute:= TRUE,
		i_bAdr:= q_stStatus.bAdr,
		i_bLen:= 0,
		i_bCmd:= 16#65,
		i_abTxData := abTxData,
		i_tTimeOut:= i_tTimeOut,
		iq_stSerialRXBuffer:= iq_stSerialRXBuffer,
		iq_stSerialTXBuffer:= iq_stSerialTXBuffer
		);
	IF fbSensirionTransaction.q_xError THEN
		q_asResult[iResultIndex] := CONCAT('in Step 400 serial transaction failed with message: ', fbSensirionTransaction.q_sResult);
		iResultIndex := iResultIndex +1;
		iStep := 9000;
	ELSIF fbSensirionTransaction.q_xDone THEN
		tonCommandDelay(IN:=fbSensirionTransaction.q_xDone, PT:=T#200MS);
		IF tonCommandDelay.Q THEN
			q_asResult[iResultIndex] := 'Device reset command sent';
			iResultIndex := iResultIndex +1;	
			iStep:=8000;
			xInitComplete := FALSE;
			fbSensirionTransaction( i_xExecute:= FALSE, iq_stSerialRXBuffer:= iq_stSerialRXBuffer, iq_stSerialTXBuffer:= iq_stSerialTXBuffer );  (* reset *)
		END_IF
	END_IF	
	
	
	20: //Start continuous measurement
	abTxData[1]:=0;
	abTxData[2]:=0;
		fbSensirionTransaction(
			i_xExecute:= TRUE,
			i_bAdr:= q_stStatus.bAdr,
			i_bLen:= 2,
			i_bCmd:= 16#33,
			i_abTxData := abTxData,
			i_tTimeOut:= i_tTimeOut,
			iq_stSerialRXBuffer:= iq_stSerialRXBuffer,
			iq_stSerialTXBuffer:= iq_stSerialTXBuffer
			);
		IF fbSensirionTransaction.q_xError THEN
			q_asResult[iResultIndex] := CONCAT('in Step 20 serial transaction failed with message: ', fbSensirionTransaction.q_sResult);
			iResultIndex := iResultIndex +1;
			iStep := 9000;
		ELSIF fbSensirionTransaction.q_xDone THEN
			tonCommandDelay(IN:=fbSensirionTransaction.q_xDone, PT:=T#250MS);
			IF tonCommandDelay.Q THEN	
				(* No response, completed transaction confirmed by a response*)
				iStep := 21;	
				q_asResult[iResultIndex] := CONCAT('Sent start measurement command', fbSensirionTransaction.q_sResult);
				iResultIndex := iResultIndex +1;
				fbSensirionTransaction( i_xExecute:= FALSE, iq_stSerialRXBuffer:= iq_stSerialRXBuffer, iq_stSerialTXBuffer:= iq_stSerialTXBuffer );  (* reset *)
			END_IF
		END_IF
		
	21: //Check sensor status
	fbSensirionTransaction(
		i_xExecute:= TRUE,
		i_bAdr:= q_stStatus.bAdr,
		i_bLen:= 0,
		i_bCmd:= 16#30,
		i_abTxData := abTxData,
		i_tTimeOut:= i_tTimeOut,
		iq_stSerialRXBuffer:= iq_stSerialRXBuffer,
		iq_stSerialTXBuffer:= iq_stSerialTXBuffer
		);
	IF fbSensirionTransaction.q_xError THEN
		q_asResult[iResultIndex] := CONCAT('in Step 21 serial transaction failed with message: ', fbSensirionTransaction.q_sResult);
		iResultIndex := iResultIndex +1;
		iStep := 9000;
	ELSIF fbSensirionTransaction.q_xDone THEN
		(* The status measurement is available at the rx data here *)
		IF fbSensirionTransaction.q_iRxLen > 0 THEN
			IF UDINT_TO_BOOL(MEMCPY(destAddr:=ADR(q_stStatus.bStatus), srcAddr:=ADR(fbSensirionTransaction.q_baRxData), n:=1)) THEN
				IF q_stStatus.bStatus.1 = 1 THEN
					iStep :=30;
					xInitComplete	:= TRUE;
					q_asResult[iResultIndex] := 'Init success, sensor is measuring.';
					iResultIndex := iResultIndex +1;
					fbSensirionTransaction( i_xExecute:= FALSE, iq_stSerialRXBuffer:= iq_stSerialRXBuffer, iq_stSerialTXBuffer:= iq_stSerialTXBuffer );  (* reset *)
				ELSIF q_stStatus.bStatus.0 = 1 THEN
					iStep :=21; // if the sensor is busy, and not yet measuring, perhaps we try again
					q_asResult[iResultIndex] := 'Sensor is busy...';
					iResultIndex := iResultIndex +1;
					fbSensirionTransaction( i_xExecute:= FALSE, iq_stSerialRXBuffer:= iq_stSerialRXBuffer, iq_stSerialTXBuffer:= iq_stSerialTXBuffer );  (* reset *)					
				ELSE
					iStep := 9000;
					q_asResult[iResultIndex +1] := 'Failed to start cont. measurement in step 21';
				END_IF
			ELSE
				iStep := 9000;
				q_asResult[iResultIndex] := 'Memcpy in step 21 failed';
				iResultIndex := iResultIndex +1;
			END_IF
		ELSE
			q_asResult[iResultIndex] := 'No status data returned in step 21';
			iResultIndex := iResultIndex +1;
			iStep := 9000;
		END_IF 		
	END_IF
	
	30: //Get last measurement
		tonDelay.IN:=TRUE;
		fbSensirionTransaction(
		i_xExecute:= tonDelay.Q,
		i_bAdr:= q_stStatus.bAdr,
		i_bLen:= 0,
		i_bCmd:= 16#35,
		i_abTxData := abTxData,
		i_tTimeOut:= i_tTimeOut,
		iq_stSerialRXBuffer:= iq_stSerialRXBuffer,
		iq_stSerialTXBuffer:= iq_stSerialTXBuffer
		);
	IF fbSensirionTransaction.q_xError THEN
		q_asResult[iResultIndex] := CONCAT('in Step 30 serial transaction failed with message: ', fbSensirionTransaction.q_sResult);
		iResultIndex := iResultIndex +1;
		iStep := 9000;
	ELSIF fbSensirionTransaction.q_xDone THEN	
		(* The flow measurement is available at the rx data here *)
		IF fbSensirionTransaction.q_iRxLen > 0 THEN
			IF UDINT_TO_BOOL(MEMCPY(destAddr:=ADR(q_stStatus.uiSensorOutput), srcAddr:=ADR(fbSensirionTransaction.q_baRxData), n:=2)) THEN //always 2 for the 16 bit wide integer
				q_stStatus.uiSensorOutput := WORD_TO_UINT(HOST_TO_BE16(INT_TO_WORD(q_stStatus.uiSensorOutput))); //memcpy effs up an produces a little endian number, sensirion transmits be
				IF (q_stStatus.uiSensorOutput AND 32768) = 32768 THEN
					q_stStatus.iFlowTicks := UINT_TO_INT(-1*((q_stStatus.uiSensorOutput XOR 65535) + 1));
				ELSE
					q_stStatus.iFlowTicks := UINT_TO_INT(q_stStatus.uiSensorOutput);
				END_IF
				//Conversion from int to real value using the unit
				IF ((INT_TO_WORD(iUnit) AND 16#000F)=16#0003) OR ((INT_TO_WORD(iUnit) AND 16#000F)=16#0004) THEN //lsb of iUnit is magnitude, should only be one thing
					
					q_stStatus.rFlow := ABS((INT_TO_REAL(q_stStatus.iFlowTicks)/INT_TO_REAL(iScale))*EXPT(10,-3)); //converting from nL to uL 
					
					(* Check flow readback against calibration range for OoR *)
					//calibration of 0 for precision mode, 250 nL/min - 5000 nL/min
					// calibration of 1 for extended mode, 2000 nL/min - 20000 nL/min
					IF (q_stStatus.xFMMode =0 ) THEN
						IF (ABS(q_stStatus.rFlow) < (250E-3)) THEN
							q_stStatus.iState := 2; //<OoR
						ELSIF (ABS(q_stStatus.rFlow) > (5000E-3)) THEN
							q_stStatus.iState := 1; //OoR>
						ELSE
							q_stStatus.iState := 0; //OK
						END_IF
					ELSIF (q_stStatus.xFMMode =1 ) THEN
						IF (ABS(q_stStatus.rFlow) < (2000E-3)) THEN
							q_stStatus.iState := 2; //<OoR
						ELSIF (ABS(q_stStatus.rFlow) > (20000E-3)) THEN
							q_stStatus.iState := 1; //OoR>
						ELSE
							q_stStatus.iState := 0; // OK
						END_IF
					END_IF
					
					// Limit the measured flowrate based on the calmode, note this disregards negative flow
					IF q_stStatus.xFMMode THEN
						q_stStatus.rFlow := LIMIT(0, q_stStatus.rFlow, 20000E-3);
					ELSE
						q_stStatus.rFlow := LIMIT(0, q_stStatus.rFlow, 5000E-3);
					END_IF
					
				ELSE
					iStep := 9000;
					q_asResult[iResultIndex] := 'iUnit not recognized in step 30';
					iResultIndex := iResultIndex +1;
				END_IF
				(* Stuff worked, go to 8000 *)
				iStep := 8000;
				fbSensirionTransaction( i_xExecute:= FALSE, iq_stSerialRXBuffer:= iq_stSerialRXBuffer, iq_stSerialTXBuffer:= iq_stSerialTXBuffer );  (* reset *)
				tonDelay.IN := FALSE;
			ELSE
				iStep := 9000;
				q_asResult[iResultIndex] := 'Memcpy in step 30 failed';
				iResultIndex := iResultIndex +1;
			END_IF
		ELSE
			q_asResult[iResultIndex] := 'No flow data returned';
			iResultIndex := iResultIndex +1;
			iStep := 9000;
		END_IF
	END_IF
			
	8000: (* done *)
		q_xDone := TRUE;
		IF q_asResult[iResultIndex] = '' THEN
			q_asResult[iResultIndex] := 'Success';
			iResultIndex := iResultIndex +1;
			
		END_IF
		IF  i_xExecute = FALSE THEN
			q_xDone:= FALSE;
			iStep := 0;
		END_IF
	
	9000:
		q_xTimeout := fbSensirionTransaction.q_xTimeout;
		q_xError := TRUE;
		// If we're having issues communicating we don't want to be left thinking there's a flow... even if we know it's not valid.
		q_stStatus.xFlowValid := FALSE;
		q_stStatus.iState := 3; // Flow invalid
		q_stStatus.rFlow := 0;
END_CASE

tonDelay(PT:=T#500MS);

//q_stStatus.rFlow := INT_TO_REAL(iFlow);
iStepIndex := iStepIndex +1;
aiSteps[iStepIndex]:=iStep;


q_xInitComplete := xInitComplete;

IF iStepIndex >256 THEN iStepIndex:=1; END_IF
IF iResultIndex >60 THEN iResultIndex:=1; END_IF

ACTION A_ClearTransaction:
fbSensirionTransaction( i_xExecute:= FALSE, iq_stSerialRXBuffer:= iq_stSerialRXBuffer, iq_stSerialTXBuffer:= iq_stSerialTXBuffer );  (* reset *)
END_ACTION

ACTION Get:

END_ACTION

END_FUNCTION_BLOCK

// ---- POUs/Helpers/FB_ShiftByteArray.TcPOU
FUNCTION_BLOCK FB_ShiftByteArray
VAR_INPUT
	ptArray	:	POINTER TO BYTE;
	iSize	:	INT;
	iCurrIndex	:	INT;
	iMessageLen	:	INT;
	iShift		:	INT;
	
END_VAR
VAR_OUTPUT
	q_xError	:	BOOL;
END_VAR
VAR
	howbig	: UINT;
END_VAR

howbig := sizeof(ptArray^);
// Clear error bit
q_xError := FALSE;
IF iMessageLen = iCurrIndex THEN
	//Dont do a damn thing
	;
// Check the remaining length and shift amount summed is not greater than the total array width.
ELSIF iSize < (iMessageLen - iCurrIndex) + iShift THEN
	q_xError := TRUE;
ELSE// MEMMOVE from 1+ the current index to the remaining length by the shift amount
	IF MEMMOVE(srcAddr:=(ptArray + iCurrIndex + 1), destAddr:=(ptArray + iCurrIndex + 1 + iShift), n:=(iMessageLen + 1 - iCurrIndex)) =0 THEN
		q_xError := TRUE;
	END_IF
END_IF

END_FUNCTION_BLOCK

// ---- POUs/p_AutoWash.TcPOU
ROGRAM p_AutoWash
VAR

	

END_VAR

// ---- POUs/p_CoolerShaker.TcPOU
ROGRAM p_CoolerShaker
VAR
	
afbTECDriver	:	ARRAY[1..3] OF FB_TECDriver;

	index: INT :=1 ;
END_VAR


stTECCtrl[1].sAddress := '01'; //62 is 98 in hex which is default address
stTECCtrl[2].sAddress := '02';
stTECCtrl[3].sAddress := '62';

stTECCtrl[1].diTempSetpoint := 30; //98 in hex which is default address
stTECCtrl[2].diTempSetpoint := 30;
stTECCtrl[3].diTempSetpoint := 30;

afbTECDriver[index](
	i_xExecute:= TRUE,
	i_tTimeOut:= t#1s,
	i_stControl:= stTECCtrl[index],
	iq_stSerialRXBuffer:= SerialRXBuffer_CoolerShakerTEC,
	iq_stSerialTXBuffer:= SerialTXBuffer_CoolerShakerTEC,
	q_stStatus=>stTECStatus[index]);

IF afbTECDriver[index].q_xDone OR
	afbTECDriver[index].q_xError OR
	afbTECDriver[index].q_xTimeout THEN
	(* reset function for next time *)
	afbTECDriver[index](i_xExecute:=FALSE, iq_stSerialRXBuffer:= SerialRXBuffer_CoolerShakerTEC, iq_stSerialTXBuffer:=  SerialTXBuffer_CoolerShakerTEC);
	
	index := index + 1;
	IF index > 2 THEN index := 1; END_IF
	
END_IF

// ---- POUs/TEC/FB_TECDriver.TcPOU
FUNCTION_BLOCK FB_TECDriver

VAR_INPUT
	i_xExecute				: BOOL;					(* rising edge execute *)
	i_tTimeOut				: TIME := t#10s;  		(* Maximum wait time for reply *)
	i_stControl				: ST_TECControl;
END_VAR
VAR_OUTPUT
	q_xDone					: BOOL;
	q_xError				: BOOL;
	q_xWarning				: BOOL;					(* set in the event of an unexpected reply *)
	q_xTimeout				: BOOL;
	q_sResult				: STRING(255);
	q_sLastSentString		: ARRAY[1..40] OF STRING;				(* Last String Sent to Serial Device - for debugging *)
	q_sLastReceivedString	: ARRAY[1..40] OF STRING;				(* Last String Received from Serial Device - for debugging *)
	q_stStatus				: ST_TECStatus;
END_VAR
VAR_IN_OUT
	iq_stSerialRXBuffer 	: ComBuffer;
	iq_stSerialTXBuffer 	: ComBuffer;
END_VAR
VAR
	rtExecute				: R_TRIG;
	iStep					: INT;
	sSendData				: STRING;
	fbTECTransaction		: FB_TECTransaction;
	(*fbFormatString			: FB_FormatString;*)
	(*fbSplit					: FB_Split255;*)
	asReplyFields			: ARRAY[1..20] OF T_MaxString;
	wChecksum: WORD;
	rtStartIntegration: R_TRIG;
	rtEndReset: R_TRIG;

	sWorking: STRING;
	strResponseExpected: STRING;
	diWorking	:	DINT;
END_VAR

(* This function block performs serial communication with a TC-36-25 TEC Driver *)

(* rising edge trigger *)
rtExecute(CLK:= i_xExecute);
IF rtExecute.Q  THEN
	q_xDone	:= FALSE;
	q_xError := FALSE;
	q_xWarning := FALSE;
	q_xTimeout := FALSE;
	q_sResult:= '';
	fbTECTransaction( i_xExecute:= FALSE, iq_stSerialRXBuffer:= iq_stSerialRXBuffer, iq_stSerialTXBuffer:= iq_stSerialTXBuffer );  (* reset *)
	
	iStep := 10;
END_IF

CASE iStep OF
	0: (* idle *)
		;

	10: (* Get Current Temperature *)
		fbTECTransaction(
			i_xExecute:= TRUE,
			i_sAddress:=i_stControl.sAddress,
			i_sCmd:= '01',
			i_diParameter := 0,
			i_tTimeOut:= i_tTimeOut,
			iq_stSerialRXBuffer:= iq_stSerialRXBuffer,
			iq_stSerialTXBuffer:= iq_stSerialTXBuffer,
			i_CmdFlag :=FALSE);
			
		IF fbTECTransaction.q_xError THEN
			q_sResult := CONCAT('in Step 10 serial transaction failed with message: ', fbTECTransaction.q_sResult);
			iStep := 9000;
		ELSIF fbTECTransaction.q_xDone THEN
			q_stStatus.sReply := fbTECTransaction.q_sResponseData;
			sWorking :=LEFT(q_stStatus.sReply, 8);
			sWorking := CONCAT('16#', sWorking);
			q_stStatus.diTemp1 := STRING_TO_DINT(sWorking);
			fbTECTransaction( i_xExecute:= FALSE, iq_stSerialRXBuffer:= iq_stSerialRXBuffer, iq_stSerialTXBuffer:= iq_stSerialTXBuffer, i_CmdFlag :=FALSE);  (* reset *)
			iStep := 20;
			
		END_IF
	20: (* Read setpoint *)
		fbTECTransaction(
			i_xExecute:= TRUE,
			i_sAddress:=i_stControl.sAddress,
			i_sCmd:= '03', // command 
			i_diParameter := 0, // always zero for query
			i_tTimeOut:= i_tTimeOut,
			iq_stSerialRXBuffer:= iq_stSerialRXBuffer,
			iq_stSerialTXBuffer:= iq_stSerialTXBuffer,
			i_CmdFlag :=FALSE);
			
		IF fbTECTransaction.q_xError THEN
			q_sResult := CONCAT('in Step 20 serial transaction failed with message: ', fbTECTransaction.q_sResult);
			iStep := 9000;
		ELSIF fbTECTransaction.q_xDone THEN
			q_stStatus.sReply := fbTECTransaction.q_sResponseData;
			sWorking :=LEFT(q_stStatus.sReply, 8);
			sWorking := CONCAT('16#', sWorking);
			q_stStatus.diSetPoint := STRING_TO_DINT(sWorking);
			fbTECTransaction( i_xExecute:= FALSE, iq_stSerialRXBuffer:= iq_stSerialRXBuffer, iq_stSerialTXBuffer:= iq_stSerialTXBuffer, i_CmdFlag :=FALSE);  (* reset *)
			iStep := 25;
		END_IF
		
	25: (* Read output ON/OFF *)
		fbTECTransaction(
			i_xExecute:= TRUE,
			i_sAddress:=i_stControl.sAddress,
			i_sCmd:= '46', // command 
			i_diParameter := 0, // always zero for query
			i_tTimeOut:= i_tTimeOut,
			iq_stSerialRXBuffer:= iq_stSerialRXBuffer,
			iq_stSerialTXBuffer:= iq_stSerialTXBuffer,
			i_CmdFlag :=FALSE);
			
		IF fbTECTransaction.q_xError THEN
			q_sResult := CONCAT('in Step 25 serial transaction failed with message: ', fbTECTransaction.q_sResult);
			iStep := 9000;
		ELSIF fbTECTransaction.q_xDone THEN
			q_stStatus.sReply := fbTECTransaction.q_sResponseData;
			sWorking :=LEFT(q_stStatus.sReply, 8);
			sWorking := CONCAT('16#', sWorking);
			diWorking := STRING_TO_DINT(sWorking);
			q_stStatus.xOutputOn := DINT_TO_BOOL(diWorking);
			A_ResetTransaction();
			iStep := 30;
		END_IF
	
	30: (* Read the alarm status *)
		fbTECTransaction(
			i_xExecute:= TRUE,
			i_sAddress:=i_stControl.sAddress,
			i_sCmd:= '05', // command 
			i_diParameter := 0, // always zero for query
			i_tTimeOut:= i_tTimeOut,
			iq_stSerialRXBuffer:= iq_stSerialRXBuffer,
			iq_stSerialTXBuffer:= iq_stSerialTXBuffer,
			i_CmdFlag :=FALSE);
			
		IF fbTECTransaction.q_xError THEN
			q_sResult := CONCAT('in Step 10 serial transaction failed with message: ', fbTECTransaction.q_sResult);
			iStep := 9000;
		ELSIF fbTECTransaction.q_xDone THEN
			q_stStatus.sReply := fbTECTransaction.q_sResponseData;
			sWorking :=LEFT(q_stStatus.sReply, 8);
			sWorking := CONCAT('16#', sWorking);
			diWorking := STRING_TO_DINT(sWorking);
			
			//Alarm assignment
			q_stStatus.xHiTemp	:=	diWorking.0;
			q_stStatus.xLoTemp	:=	diWorking.1;
			q_stStatus.xLoTemp	:=	diWorking.2;
			q_stStatus.xOverCurrent	:=	diWorking.3;
			q_stStatus.xOpenInput1	:=	diWorking.4;
			q_stStatus.xOpenInput2	:=	diWorking.5;
			q_stStatus.xDriverLowVoltage	:=	diWorking.6;
			
			fbTECTransaction( i_xExecute:= FALSE, iq_stSerialRXBuffer:= iq_stSerialRXBuffer, iq_stSerialTXBuffer:= iq_stSerialTXBuffer, i_CmdFlag :=FALSE);  (* reset *)
			iStep := 40;
		END_IF
		
	40: (* Output Power *)
		fbTECTransaction(
			i_xExecute:= TRUE,
			i_sAddress:=i_stControl.sAddress,
			i_sCmd:= '02', // command 
			i_diParameter := 0, // always zero for query
			i_tTimeOut:= i_tTimeOut,
			iq_stSerialRXBuffer:= iq_stSerialRXBuffer,
			iq_stSerialTXBuffer:= iq_stSerialTXBuffer,
			i_CmdFlag :=FALSE);
			
		IF fbTECTransaction.q_xError THEN
			q_sResult := CONCAT('in Step 10 serial transaction failed with message: ', fbTECTransaction.q_sResult);
			iStep := 9000;
		ELSIF fbTECTransaction.q_xDone THEN
			q_stStatus.sReply := fbTECTransaction.q_sResponseData;
			sWorking :=LEFT(q_stStatus.sReply, 8);
			sWorking := CONCAT('16#', sWorking);
			diWorking := STRING_TO_DINT(sWorking);
			
			q_stStatus.diPercentOut := (diWorking/511)*100; //in percentage
			
			fbTECTransaction( i_xExecute:= FALSE, iq_stSerialRXBuffer:= iq_stSerialRXBuffer, iq_stSerialTXBuffer:= iq_stSerialTXBuffer, i_CmdFlag :=FALSE);  (* reset *)
			iStep := 5000;
		END_IF

	5000: (* Change Setpoint *)
		IF q_stStatus.diSetpoint <> i_stControl.diTempSetpoint THEN

			fbTECTransaction(
				i_xExecute:= TRUE,
				i_sAddress:=i_stControl.sAddress,
				i_sCmd:= '1c', // command 
				i_diParameter := i_stControl.diTempSetpoint,
				i_tTimeOut:= i_tTimeOut,
				iq_stSerialRXBuffer:= iq_stSerialRXBuffer,
				iq_stSerialTXBuffer:= iq_stSerialTXBuffer,
				i_CmdFlag :=TRUE);
			IF fbTECTransaction.q_xError THEN
				q_sResult := CONCAT('in Step 5000 serial transaction failed with message: ', fbTECTransaction.q_sResult);
				iStep := 9000;
			ELSIF fbTECTransaction.q_xDone THEN
				fbTECTransaction(
					 i_xExecute:= FALSE,
					iq_stSerialRXBuffer:= iq_stSerialRXBuffer,
					iq_stSerialTXBuffer:= iq_stSerialTXBuffer,
					i_CmdFlag:=FALSE );  (* reset *)
				iStep := 5010;
			END_IF
		ELSE
			iStep := 5010;
		END_IF
		
	5010: (* Output ON/OFF *)
		IF q_stStatus.xOutputOn <> i_stControl.xOutputOn THEN

			fbTECTransaction(
				i_xExecute:= TRUE,
				i_sAddress:=i_stControl.sAddress,
				i_sCmd:= '2d', // command 
				i_diParameter := BOOL_TO_DINT(i_stControl.xOutputOn),
				i_tTimeOut:= i_tTimeOut,
				iq_stSerialRXBuffer:= iq_stSerialRXBuffer,
				iq_stSerialTXBuffer:= iq_stSerialTXBuffer,
				i_CmdFlag :=TRUE);
			IF fbTECTransaction.q_xError THEN
				q_sResult := CONCAT('in Step 5010 serial transaction failed with message: ', fbTECTransaction.q_sResult);
				iStep := 9000;
			ELSIF fbTECTransaction.q_xDone THEN
				fbTECTransaction(
					 i_xExecute:= FALSE,
					iq_stSerialRXBuffer:= iq_stSerialRXBuffer,
					iq_stSerialTXBuffer:= iq_stSerialTXBuffer,
					i_CmdFlag:=FALSE );  (* reset *)
				iStep := 8000;
			END_IF
		ELSE
			iStep := 8000;
		END_IF


	8000: (* done *)
		q_xDone := TRUE;
		IF q_sResult = '' THEN
			q_sResult := 'Success';
			q_stStatus.xStatusValid := TRUE;
		END_IF
		IF  i_xExecute = FALSE THEN
			q_xDone:= FALSE;
			iStep := 0;
		END_IF

	9000:
		_A_ClearStatus();
		q_xTimeout := fbTECTransaction.q_xTimeout;
		q_xError := TRUE;
		q_stStatus.xStatusValid := FALSE;
		

END_CASE

q_sLastSentString := fbTECTransaction.q_sLastSentString;
q_sLastReceivedString := fbTECTransaction.q_sLastReceivedString;

ACTION A_ResetTransaction:
fbTECTransaction( i_xExecute:= FALSE, iq_stSerialRXBuffer:= iq_stSerialRXBuffer, iq_stSerialTXBuffer:= iq_stSerialTXBuffer, i_CmdFlag :=FALSE);  (* reset *)
END_ACTION

ACTION _A_ClearStatus:
q_stStatus.sReply := '';
END_ACTION

END_FUNCTION_BLOCK

// ---- POUs/p_Shakers.TcPOU
ROGRAM p_Shakers
VAR
END_VAR

// ---- POUs/p_VacGaugeSup.TcPOU
PROGRAM p_VacGaugeSup 

VAR

	
	
END_VAR

END_PROGRAM

// ---- POUs/Regulators/FB_Regulator.TcPOU
FUNCTION_BLOCK FB_Regulator
VAR_INPUT
	iI: INT;
	lrVelocity	:	LREAL := 360;
END_VAR
VAR_OUTPUT
q_asResult: ARRAY [1..20] OF STRING;
q_xError	:	BOOL;
END_VAR
VAR_IN_OUT
	iq_stRegulator	:	ST_Regulator;
END_VAR
VAR
	

mcPower	:	MC_Power;
mcSetHome	:	MC_SetPosition;
mcReset	:	MC_Reset;
mcMoveAbsolute : ARRAY[1..2] OF MC_MoveAbsolute;
mcStatus : MC_ReadStatus;

mcHalt	:	MC_Halt;

	iPressDiff: INT;
	iTolerance: INT := 50;
	xMoveOK: BOOL;
	iStep: INT;
	
	indexResult: INT := 1;
	
	xInitComplete	:	BOOL := FALSE;
	
	ftBackToAuto	:	F_TRIG;
	iPercSPOld: UINT;
	imcBlockIndex: INT;
	imcBlockIndexPrev : INT;
	
	rtEnable : R_TRIG;
END_VAR

(* Regulator Function Block *)
(* Alex Wallace, 2014-10-16 *)
(* Modified in 2.5.3 to remove all pressure SP  based code *)

rtEnable(CLK:=iq_stRegulator.xRegEnab);

(* Regulator Pressure Calculation *)
iq_stRegulator.wInPress := LIMIT(0, F_rPressure(iRawVoltage := iq_stRegulator.i_iRawInPress), 10000);
iq_stRegulator.wOutPress := LIMIT(0, F_rPressure(iRawVoltage := iq_stRegulator.i_iRawOutPress), 10000);


(* Basic regulator interlocking *)


(* Check for regulator enable *)
xMoveOK := iq_stRegulator.xRegEnab;
IF NOT xMoveOK THEN
	(*iq_stRegulator.wPressSP := 0; not preferred *)
	iq_stRegulator.xRegEnab := FALSE;
	(* add motor error here *)
END_IF

IF q_xError THEN
	iStep := 9000;
ELSIF rtEnable.Q THEN
	xInitComplete := FALSE;
	iStep := 10;
ELSIF xInitComplete THEN
	iStep := 3000;
END_IF


CASE iStep OF
	0: iStep := 10;
	10:
	(* Start by initializing the motor axis *)
	mcPower.Enable := TRUE;
	iq_stRegulator.lrUpperLimPos := 2887;
	IF mcPower.Status THEN
		xInitComplete := TRUE;
		q_asResult[indexResult] := 'Motor init success';
		indexResult := indexResult + 1;
		iStep := 3000;
	ELSIF mcPower.Error THEN
		mcPower.Enable := FALSE;
		iStep := 9000;
		q_xError	:=	TRUE;
		q_asResult[indexResult] := CONCAT('Initilizing regulator motor in step 10 failed with error code: ', UDINT_TO_STRING(mcPower.ErrorID));
		indexResult := indexResult +1;
	END_IF
		
	//Knob controls
	3000:
	
	IF iq_stRegulator.i_iPercSP <> iPercSPOld  AND xMoveOK THEN
		mcMoveAbsolute[imcBlockIndex].Execute := FALSE;
		imcBlockIndex := imcBlockIndex + 1;
		IF imcBlockIndex >2 THEN imcBlockIndex := 1; END_IF
		mcMoveAbsolute[imcBlockIndex].Position := LIMIT(0, UINT_TO_LREAL(iq_stRegulator.i_iPercSP) * iq_stRegulator.lrUpperLimPos/65535, MAX(iq_stRegulator.lrUpperLimPos,1));
		mcMoveAbsolute[imcBlockIndex].Execute := TRUE;
		iPercSPOld := iq_stRegulator.i_iPercSP;
	ELSIF mcMoveAbsolute[imcBlockIndex].Done or mcMoveAbsolute[imcBlockIndex].CommandAborted or mcMoveAbsolute[imcBlockIndex].Busy or mcMoveAbsolute[imcBlockIndex].Error THEN
		mcMoveAbsolute[imcBlockIndex].Execute := FALSE;
	END_IF
	
	9000:
	(* Error *)
	mcReset.Execute := iq_stRegulator.xRegEnab;
	IF mcReset.Done THEN
		q_xError := FALSE;
		mcReset.Execute := FALSE;
		iStep:=10;
	END_IF
	
END_CASE

//Reset the debugging index
IF indexResult > 20 THEN indexResult := 1; END_IF

(* Regulator Percentage Open *)
(* Calculate the regulator percentage open, based on 6.5 turns to fully open *)

iq_stRegulator.wPercentageOpen := LREAL_TO_WORD( (iq_stRegulator.stRegulatorMotor.NcToPlc.ActPos / MAX(iq_stRegulator.lrUpperLimPos,1))*100);

(* Run the mc blocks *)
iq_stRegulator.stRegulatorMotor();
ActPower();

mcSetHome(Execute:=NOT(iq_stRegulator.xRegLoLS) AND iq_stRegulator.stRegulatorMotor.Status.StandStill, Axis:=iq_stRegulator.stRegulatorMotor, Position:=0, Mode:=FALSE);
IF NOT iq_stRegulator.xRegHiLS THEN iq_stRegulator.lrUpperLimPos := iq_stRegulator.stRegulatorMotor.NcToPlc.ActPos; END_IF
mcReset(Axis:=iq_stRegulator.stRegulatorMotor);

FOR iI := 1 TO 2 DO
mcMoveAbsolute[iI](Axis := iq_stRegulator.stRegulatorMotor, Velocity:=iq_stRegulator.lrVelocity, BufferMode:=MC_Aborting);
END_FOR

IF mcMoveAbsolute[1].Error OR mcMoveAbsolute[2].Error THEN
	q_xError	:=	TRUE;
	mcMoveAbsolute[1].Execute := FALSE;
	mcMoveAbsolute[2].Execute := FALSE;
	q_asResult[indexResult] := 'Error occured with motion blocks';
	indexResult := indexResult +1;
ELSIF mcPower.Error THEN
	q_xError := TRUE;
	q_asResult[indexResult] := concat('mcPower block error: ', UDINT_TO_STRING(mcPower.ErrorID));
END_IF

ACTION ActPower:
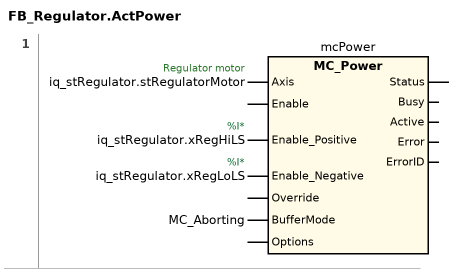
// NETWORK 1
//   iq_stRegulator.stRegulatorMotor: Regulator motor
//   iq_stRegulator.xRegHiLS: AT %I*
//   iq_stRegulator.xRegLoLS: AT %I*
mcPower(
    Axis := iq_stRegulator.stRegulatorMotor,
    Enable_Positive := iq_stRegulator.xRegHiLS,
    Enable_Negative := iq_stRegulator.xRegLoLS,
    BufferMode := MC_Aborting); // MC_Power
END_ACTION

END_FUNCTION_BLOCK

// ---- POUs/SerialTxRx.TcPOU
PROGRAM SerialTxRx
VAR
	
	fbSerialLineControl_SelectorVici: SerialLineControl;
	fbSerialLineControl_Selector2Vici: SerialLineControl;
	fbSerialLineControl_SelectorFlwMtr: SerialLineControl;
	fbSerialLineControl_Selector2FlwMtr: SerialLineControl;
	fbSerialLineControl_CoolerShakerTEC: SerialLineControl;
	


END_VAR



fbSerialLineControl_SelectorVici(
	Mode:= SERIALLINEMODE_EL6_22B (*SERIALLINEMODE_KL6_22B_STANDARD*),
	pComIn:= ADR(stComIn_SelB2P2),
	pComOut:=ADR(stComOut_SelB2P2) ,
	SizeComIn:= SIZEOF(stComIn_SelB2P2),
	TxBuffer:= SerialTXBuffer_SelVici,
	RxBuffer:= SerialRXBuffer_SelVici,
	Error=> ,
	ErrorID=> );
	
	(* Optional expansion for extra selector box *)
fbSerialLineControl_Selector2Vici(
	Mode:= SERIALLINEMODE_EL6_22B (*SERIALLINEMODE_KL6_22B_STANDARD*),
	pComIn:= ADR(stComIn_Sel2B2P2),
	pComOut:=ADR(stComOut_Sel2B2P2) ,
	SizeComIn:= SIZEOF(stComIn_Sel2B2P2),
	TxBuffer:= SerialTXBuffer_Sel2Vici,
	RxBuffer:= SerialRXBuffer_Sel2Vici,
	Error=> ,
	ErrorID=> );
	
	fbSerialLineControl_SelectorFlwMtr(
	Mode:= SERIALLINEMODE_EL6_22B (*SERIALLINEMODE_KL6_22B_STANDARD*),
	pComIn:= ADR(stComIn_SelB2P1),
	pComOut:=ADR(stComOut_SelB2P1) ,
	SizeComIn:= SIZEOF(stComIn_SelB2P1),
	TxBuffer:= SerialTXBuffer_SelFlwMtr,
	RxBuffer:= SerialRXBuffer_SelFlwMtr,
	Error=> ,
	ErrorID=> );
	
fbSerialLineControl_Selector2FlwMtr(
	Mode:= SERIALLINEMODE_EL6_22B (*SERIALLINEMODE_KL6_22B_STANDARD*),
	pComIn:= ADR(stComIn_Sel2B2P1),
	pComOut:=ADR(stComOut_Sel2B2P1) ,
	SizeComIn:= SIZEOF(stComIn_Sel2B2P1),
	TxBuffer:= SerialTXBuffer_Sel2FlwMtr,
	RxBuffer:= SerialRXBuffer_Sel2FlwMtr,
	Error=> ,
	ErrorID=> );

END_PROGRAM
